KUKA KRL program: EPS_2_251806_MH47A_A_20260213065144.src

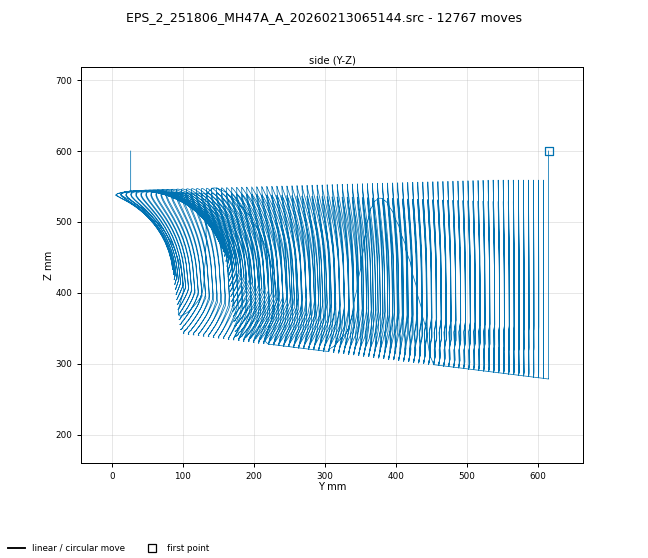
[picture p0: tool path of EPS_2_251806_MH47A_A_20260213065144.src, 12767 of 12769 moves have a stored position in this frame; points joined in program order, loops and branches not executed]
&ACCESS RVP
&REL 4
&COMMENT QRS 19112012
&PARAM EDITMASK = *
DEF PART()
EXT BAS (BAS_COMMAND :IN,REAL :IN )
INT I
BAS (#INITMOV,0 )

;KUKA QRS Post kuka4.cps  Date:22-06-2017 !

File_ID=3034

QRS_PRE_INIT()

;Init var - Until changes are made in qrs_pre_init
Outlet_Square_prg=0
Inlet_1_Square_prg=0
Inlet_2_Square_prg=0
Inlet_3_Square_prg=0
Inlet_4_Square_prg=0
Inlet_5_Square_prg=0

Outlet_1={X 0.000, Y 535.490, Z 458.500, B 0.000, E1 0.000 }
Inlet_1={X 0.000, Y 537.630, Z 428.500, B 0.000, E1 194.000 }
Outlet_1_type=201
Inlet_1_type=201
;QRS#1=Sidecore dimensions
;QRS#2=200-8" PVC SDR 35
;QRS#3=200-8" PVC SDR 35
;QRS#4=
;QRS#5=
;QRS#6=
;QRS#7=
;QRS#8=
;QRS#9=12-08 PSX
;QRS#10=12-08 PSX
;QRS#11=
;QRS#12=
;QRS#13=
;QRS#14=
;QRS#15=
;QRS#16=1220x127x838 2,75'
;QRS#17=EPS Height
;QRS#18=559
;QRS#19=*
;QRS#20= UPDATED VERSION 22-06-2017
;QRS#21=*
Outlet_Square=0100
Inlet_1_Square=0100
Inlet_2_Square=0
Inlet_3_Square=0
Inlet_4_Square=0
Inlet_5_Square=0
Mill_Square=1
Outlet_Square_Prg=204
Inlet_1_Square_prg=204

QRS_INIT()

$ADVANCE=5

; T1
PTP {E1 173.619,E2 173.619}
PTP {X 0,Y 615.497,A -85,B 0,C 180,E1 173.619,E2 173.619,E3 0,E4 0,E5 0,E6 0}
QRS_SPEED_INIT()
LIN {X 0,Y 615.497,Z 600,A -85,B 0,C 180,E1 173.619,E2 173.619,E3 0,E4 0,E5 0,E6 0} C_VEL
LIN {X 0,Y 615.497,Z 288.877,A -85,B 0,C 180,E1 173.619,E2 173.619} C_VEL
LIN {X 0,Y 615.497,Z 280.697,A -85,B 0,C 180,E1 173.619,E2 173.619} C_VEL
LIN {X 0,Y 615.476,Z 278.697,A -85,B 0,C 180,E1 173.433,E2 173.433} C_VEL
LIN {X 0,Y 615.451,Z 278.69,A -85,B 0,C 180,E1 170.801,E2 170.801} C_VEL
LIN {X 0,Y 615.482,Z 278.683,A -85,B 0,C 180,E1 168.139,E2 168.139} C_VEL
LIN {X 0,Y 615.489,Z 278.698,A -85,B 0,C 180,E1 165.451,E2 165.451} C_VEL
LIN {X 0,Y 615.453,Z 278.694,A -85,B 0,C 180,E1 162.729,E2 162.729} C_VEL
LIN {X 0,Y 615.455,Z 278.693,A -85,B 0,C 180,E1 160.661,E2 160.661} C_VEL
LIN {X 0,Y 615.455,Z 278.693,A -85,B 0,C 180,E1 158.567,E2 158.567} C_VEL
LIN {X 0,Y 615.458,Z 278.687,A -85,B 0,C 180,E1 155.998,E2 155.998} C_VEL
LIN {X 0,Y 615.483,Z 278.683,A -85,B 0,C 180,E1 153.556,E2 153.556} C_VEL
LIN {X 0,Y 615.475,Z 278.699,A -85,B 0,C 180,E1 150.593,E2 150.593} C_VEL
LIN {X 0,Y 615.462,Z 278.695,A -85,B 0,C 180,E1 148.313,E2 148.313} C_VEL
LIN {X 0,Y 615.451,Z 278.692,A -85,B 0,C 180,E1 145.976,E2 145.976} C_VEL
LIN {X 0,Y 615.455,Z 278.688,A -85,B 0,C 180,E1 143.573,E2 143.573} C_VEL
LIN {X 0,Y 615.494,Z 278.683,A -85,B 0,C 180,E1 140.938,E2 140.938} C_VEL
LIN {X 0,Y 615.491,Z 278.693,A -85,B 0,C 180,E1 138.527,E2 138.527} C_VEL
LIN {X 0,Y 615.46,Z 278.696,A -85,B 0,C 180,E1 135.848,E2 135.848} C_VEL
LIN {X 0,Y 615.452,Z 278.689,A -85,B 0,C 180,E1 133.248,E2 133.248} C_VEL
LIN {X 0,Y 615.488,Z 278.683,A -85,B 0,C 180,E1 130.607,E2 130.607} C_VEL
LIN {X 0,Y 615.487,Z 278.698,A -85,B 0,C 180,E1 128.012,E2 128.012} C_VEL
LIN {X 0,Y 615.477,Z 278.698,A -85,B 0,C 180,E1 125.617,E2 125.617} C_VEL
LIN {X 0,Y 615.455,Z 278.694,A -85,B 0,C 180,E1 123.239,E2 123.239} C_VEL
LIN {X 0,Y 615.447,Z 278.691,A -85,B 0,C 180,E1 120.922,E2 120.922} C_VEL
LIN {X 0,Y 615.462,Z 278.686,A -85,B 0,C 180,E1 118.446,E2 118.446} C_VEL
LIN {X 0,Y 615.491,Z 278.696,A -85,B 0,C 180,E1 115.57,E2 115.57} C_VEL
LIN {X 0,Y 615.455,Z 278.694,A -85,B 0,C 180,E1 112.846,E2 112.846} C_VEL
LIN {X 0,Y 615.449,Z 278.691,A -85,B 0,C 180,E1 110.548,E2 110.548} C_VEL
LIN {X 0,Y 615.47,Z 278.685,A -85,B 0,C 180,E1 107.958,E2 107.958} C_VEL
LIN {X 0,Y 615.493,Z 278.694,A -85,B 0,C 180,E1 105.226,E2 105.226} C_VEL
LIN {X 0,Y 615.459,Z 278.695,A -85,B 0,C 180,E1 102.531,E2 102.531} C_VEL
LIN {X 0,Y 615.465,Z 278.696,A -85,B 0,C 180,E1 100.528,E2 100.528} C_VEL
LIN {X 0,Y 615.472,Z 278.697,A -85,B 0,C 180,E1 98.537,E2 98.537} C_VEL
LIN {X 0,Y 615.448,Z 278.69,A -85,B 0,C 180,E1 95.899,E2 95.899} C_VEL
LIN {X 0,Y 615.489,Z 278.782,A -85,B 0,C 180,E1 95.201,E2 95.201} C_VEL
LIN {X 0,Y 615.493,Z 296.487,A -85,B 0,C 180,E1 92.291,E2 92.291} C_VEL
LIN {X 0,Y 615.474,Z 313.65,A -85,B 0,C 180,E1 89.51,E2 89.51} C_VEL
LIN {X 0,Y 615.497,Z 317.957,A -85,B 0,C 180,E1 88.815,E2 88.815} C_VEL
LIN {X 0,Y 615.476,Z 424.728,A -85,B 0,C 180,E1 87.546,E2 87.546} C_VEL
LIN {X 0,Y 615.474,Z 437.838,A -85,B 0,C 180,E1 87.26,E2 87.26} C_VEL
LIN {X 0,Y 615.498,Z 450.38,A -85,B 0,C 180,E1 86.851,E2 86.851} C_VEL
LIN {X 0,Y 615.484,Z 462.433,A -85,B 0,C 180,E1 86.318,E2 86.318} C_VEL
LIN {X 0,Y 615.494,Z 473.824,A -85,B 0,C 180,E1 85.662,E2 85.662} C_VEL
LIN {X 0,Y 615.499,Z 483.003,A -85,B 0,C 180,E1 85.006,E2 85.006} C_VEL
LIN {X 0,Y 615.497,Z 491.611,A -85,B 0,C 180,E1 84.267,E2 84.267} C_VEL
LIN {X 0,Y 615.494,Z 499.888,A -85,B 0,C 180,E1 83.416,E2 83.416} C_VEL
LIN {X 0,Y 615.49,Z 507.472,A -85,B 0,C 180,E1 82.455,E2 82.455} C_VEL
LIN {X 0,Y 615.496,Z 513.737,A -85,B 0,C 180,E1 81.464,E2 81.464} C_VEL
LIN {X 0,Y 615.497,Z 518.737,A -85,B 0,C 180,E1 80.471,E2 80.471} C_VEL
LIN {X 0,Y 615.497,Z 522.611,A -85,B 0,C 180,E1 79.474,E2 79.474} C_VEL
LIN {X 0,Y 615.497,Z 524.605,A -85,B 0,C 180,E1 78.808,E2 78.808} C_VEL
LIN {X 0,Y 615.495,Z 526.183,A -85,B 0,C 180,E1 78.14,E2 78.14} C_VEL
LIN {X 0,Y 615.496,Z 527.336,A -85,B 0,C 180,E1 77.471,E2 77.471} C_VEL
LIN {X 0,Y 615.495,Z 528.353,A -85,B 0,C 180,E1 76.127,E2 76.127} C_VEL
LIN {X 0,Y 615.497,Z 528.272,A -85,B 0,C 180,E1 75.452,E2 75.452} C_VEL
LIN {X 0,Y 615.494,Z 527.732,A -85,B 0,C 180,E1 74.775,E2 74.775} C_VEL
LIN {X 0,Y 615.494,Z 525.742,A -85,B 0,C 180,E1 73.567,E2 73.567} C_VEL
LIN {X 0,Y 615.496,Z 522.457,A -85,B 0,C 180,E1 72.388,E2 72.388} C_VEL
LIN {X 0,Y 615.497,Z 518.375,A -85,B 0,C 180,E1 71.355,E2 71.355} C_VEL
LIN {X 0,Y 615.497,Z 511.947,A -85,B 0,C 180,E1 70.142,E2 70.142} C_VEL
LIN {X 0,Y 615.497,Z 504.808,A -85,B 0,C 180,E1 69.095,E2 69.095} C_VEL
LIN {X 0,Y 615.499,Z 497.411,A -85,B 0,C 180,E1 68.218,E2 68.218} C_VEL
LIN {X 0,Y 615.496,Z 487.591,A -85,B 0,C 180,E1 67.28,E2 67.28} C_VEL
LIN {X 0,Y 615.493,Z 478.076,A -85,B 0,C 180,E1 66.534,E2 66.534} C_VEL
LIN {X 0,Y 615.484,Z 467.445,A -85,B 0,C 180,E1 65.86,E2 65.86} C_VEL
LIN {X 0,Y 615.494,Z 455.76,A -85,B 0,C 180,E1 65.28,E2 65.28} C_VEL
LIN {X 0,Y 615.481,Z 442.758,A -85,B 0,C 180,E1 64.794,E2 64.794} C_VEL
LIN {X 0,Y 615.472,Z 430.437,A -85,B 0,C 180,E1 64.47,E2 64.47} C_VEL
LIN {X 0,Y 615.476,Z 417.236,A -85,B 0,C 180,E1 64.262,E2 64.262} C_VEL
LIN {X 0,Y 615.496,Z 317.894,A -85,B 0,C 180,E1 63.085,E2 63.085} C_VEL
LIN {X 0,Y 615.476,Z 300.108,A -85,B 0,C 180,E1 60.207,E2 60.207} C_VEL
LIN {X 0,Y 615.495,Z 283.831,A -85,B 0,C 180,E1 57.544,E2 57.544} C_VEL
LIN {X 0,Y 615.443,Z 278.695,A -85,B 0,C 180,E1 56.69,E2 56.69} C_VEL
LIN {X 0,Y 615.442,Z 278.691,A -85,B 0,C 180,E1 54.172,E2 54.172} C_VEL
LIN {X 0,Y 615.451,Z 278.69,A -85,B 0,C 180,E1 51.93,E2 51.93} C_VEL
LIN {X 0,Y 615.49,Z 278.69,A -85,B 0,C 180,E1 49.395,E2 49.395} C_VEL
LIN {X 0,Y 615.469,Z 278.698,A -85,B 0,C 180,E1 46.755,E2 46.755} C_VEL
LIN {X 0,Y 615.431,Z 278.695,A -85,B 0,C 180,E1 44.155,E2 44.155} C_VEL
LIN {X 0,Y 615.429,Z 278.695,A -85,B 0,C 180,E1 42.075,E2 42.075} C_VEL
LIN {X 0,Y 615.429,Z 278.694,A -85,B 0,C 180,E1 39.755,E2 39.755} C_VEL
LIN {X 0,Y 615.458,Z 278.692,A -85,B 0,C 180,E1 37.244,E2 37.244} C_VEL
LIN {X 0,Y 615.498,Z 278.697,A -85,B 0,C 180,E1 34.704,E2 34.704} C_VEL
LIN {X 0,Y 615.468,Z 278.699,A -85,B 0,C 180,E1 32.33,E2 32.33} C_VEL
LIN {X 0,Y 615.421,Z 278.698,A -85,B 0,C 180,E1 29.786,E2 29.786} C_VEL
LIN {X 0,Y 615.434,Z 278.699,A -85,B 0,C 180,E1 27.918,E2 27.918} C_VEL
LIN {X 0,Y 615.418,Z 278.697,A -85,B 0,C 180,E1 25.557,E2 25.557} C_VEL
LIN {X 0,Y 615.419,Z 278.698,A -85,B 0,C 180,E1 23.559,E2 23.559} C_VEL
LIN {X 0,Y 615.415,Z 278.698,A -85,B 0,C 180,E1 21.434,E2 21.434} C_VEL
LIN {X 0,Y 615.413,Z 278.698,A -85,B 0,C 180,E1 19.34,E2 19.34} C_VEL
LIN {X 0,Y 615.411,Z 278.699,A -85,B 0,C 180,E1 17.273,E2 17.273} C_VEL
LIN {X 0,Y 615.41,Z 278.699,A -85,B 0,C 180,E1 15.228,E2 15.228} C_VEL
LIN {X 0,Y 615.411,Z 278.699,A -85,B 0,C 180,E1 13.203,E2 13.203} C_VEL
LIN {X 0,Y 615.404,Z 278.699,A -85,B 0,C 180,E1 10.853,E2 10.853} C_VEL
LIN {X 0,Y 615.415,Z 278.7,A -85,B 0,C 180,E1 9.2,E2 9.2} C_VEL
LIN {X 0,Y 615.421,Z 278.7,A -85,B 0,C 180,E1 7.216,E2 7.216} C_VEL
LIN {X 0,Y 615.43,Z 278.7,A -85,B 0,C 180,E1 5.242,E2 5.242} C_VEL
LIN {X 0,Y 615.443,Z 278.699,A -85,B 0,C 180,E1 3.273,E2 3.273} C_VEL
LIN {X 0,Y 615.406,Z 278.699,A -85,B 0,C 180,E1 0.654,E2 0.654} C_VEL
LIN {X 0,Y 615.411,Z 278.698,A -85,B 0,C 180,E1 -1.309,E2 -1.309} C_VEL
LIN {X 0,Y 615.418,Z 278.698,A -85,B 0,C 180,E1 -3.273,E2 -3.273} C_VEL
LIN {X 0,Y 615.426,Z 278.697,A -85,B 0,C 180,E1 -5.242,E2 -5.242} C_VEL
LIN {X 0,Y 615.437,Z 278.696,A -85,B 0,C 180,E1 -7.216,E2 -7.216} C_VEL
LIN {X 0,Y 615.448,Z 278.695,A -85,B 0,C 180,E1 -9.2,E2 -9.2} C_VEL
LIN {X 0,Y 615.459,Z 278.695,A -85,B 0,C 180,E1 -11.194,E2 -11.194} C_VEL
LIN {X 0,Y 615.417,Z 278.696,A -85,B 0,C 180,E1 -13.91,E2 -13.91} C_VEL
LIN {X 0,Y 615.418,Z 278.696,A -85,B 0,C 180,E1 -15.907,E2 -15.907} C_VEL
LIN {X 0,Y 615.422,Z 278.695,A -85,B 0,C 180,E1 -17.959,E2 -17.959} C_VEL
LIN {X 0,Y 615.422,Z 278.695,A -85,B 0,C 180,E1 -20.035,E2 -20.035} C_VEL
LIN {X 0,Y 615.424,Z 278.696,A -85,B 0,C 180,E1 -22.334,E2 -22.334} C_VEL
LIN {X 0,Y 615.469,Z 278.699,A -85,B 0,C 180,E1 -24.993,E2 -24.993} C_VEL
LIN {X 0,Y 615.455,Z 278.691,A -85,B 0,C 180,E1 -27.917,E2 -27.917} C_VEL
LIN {X 0,Y 615.442,Z 278.692,A -85,B 0,C 180,E1 -30.163,E2 -30.163} C_VEL
LIN {X 0,Y 615.433,Z 278.693,A -85,B 0,C 180,E1 -32.461,E2 -32.461} C_VEL
LIN {X 0,Y 615.432,Z 278.695,A -85,B 0,C 180,E1 -34.819,E2 -34.819} C_VEL
LIN {X 0,Y 615.458,Z 278.697,A -85,B 0,C 180,E1 -37.244,E2 -37.244} C_VEL
LIN {X 0,Y 615.495,Z 278.686,A -85,B 0,C 180,E1 -40.091,E2 -40.091} C_VEL
LIN {X 0,Y 615.468,Z 278.688,A -85,B 0,C 180,E1 -42.355,E2 -42.355} C_VEL
LIN {X 0,Y 615.441,Z 278.691,A -85,B 0,C 180,E1 -44.928,E2 -44.928} C_VEL
LIN {X 0,Y 615.443,Z 278.691,A -85,B 0,C 180,E1 -46.957,E2 -46.957} C_VEL
LIN {X 0,Y 615.447,Z 278.694,A -85,B 0,C 180,E1 -49.391,E2 -49.391} C_VEL
LIN {X 0,Y 615.48,Z 278.703,A -85,B 0,C 180,E1 -51.989,E2 -51.989} C_VEL
LIN {X 0,Y 615.493,Z 278.69,A -85,B 0,C 180,E1 -54.386,E2 -54.386} C_VEL
LIN {X 0,Y 615.485,Z 278.684,A -85,B 0,C 180,E1 -56.765,E2 -56.765} C_VEL
LIN {X 0,Y 615.468,Z 278.685,A -85,B 0,C 180,E1 -59.08,E2 -59.08} C_VEL
LIN {X 0,Y 615.45,Z 278.69,A -85,B 0,C 180,E1 -61.557,E2 -61.557} C_VEL
LIN {X 0,Y 615.451,Z 278.689,A -85,B 0,C 180,E1 -63.555,E2 -63.555} C_VEL
LIN {X 0,Y 615.459,Z 278.694,A -85,B 0,C 180,E1 -65.998,E2 -65.998} C_VEL
LIN {X 0,Y 615.454,Z 278.772,A -85,B 0,C 180,E1 -67.838,E2 -67.838} C_VEL
LIN {X 0,Y 615.483,Z 297.825,A -85,B 0,C 180,E1 -70.489,E2 -70.489} C_VEL
LIN {X 0,Y 615.496,Z 319.19,A -85,B 0,C 180,E1 -73.414,E2 -73.414} C_VEL
LIN {X 0,Y 615.486,Z 340.532,A -85,B 0,C 180,E1 -76.295,E2 -76.295} C_VEL
LIN {X 0,Y 615.476,Z 346.648,A -85,B 0,C 180,E1 -77.114,E2 -77.114} C_VEL
LIN {X 0,Y 615.488,Z 454.868,A -85,B 0,C 180,E1 -78.411,E2 -78.411} C_VEL
LIN {X 0,Y 615.493,Z 467.368,A -85,B 0,C 180,E1 -78.683,E2 -78.683} C_VEL
LIN {X 0,Y 615.492,Z 480.562,A -85,B 0,C 180,E1 -79.111,E2 -79.111} C_VEL
LIN {X 0,Y 615.489,Z 492.49,A -85,B 0,C 180,E1 -79.64,E2 -79.64} C_VEL
LIN {X 0,Y 615.478,Z 504.007,A -85,B 0,C 180,E1 -80.304,E2 -80.304} C_VEL
LIN {X 0,Y 615.498,Z 513.229,A -85,B 0,C 180,E1 -80.968,E2 -80.968} C_VEL
LIN {X 0,Y 615.498,Z 521.009,A -85,B 0,C 180,E1 -81.63,E2 -81.63} C_VEL
LIN {X 0,Y 615.497,Z 530.612,A -85,B 0,C 180,E1 -82.62,E2 -82.62} C_VEL
LIN {X 0,Y 615.49,Z 538.208,A -85,B 0,C 180,E1 -83.609,E2 -83.609} C_VEL
LIN {X 0,Y 615.498,Z 545.208,A -85,B 0,C 180,E1 -84.76,E2 -84.76} C_VEL
LIN {X 0,Y 615.493,Z 549.854,A -85,B 0,C 180,E1 -85.744,E2 -85.744} C_VEL
LIN {X 0,Y 615.496,Z 553.4,A -85,B 0,C 180,E1 -86.728,E2 -86.728} C_VEL
LIN {X 0,Y 615.497,Z 555.234,A -85,B 0,C 180,E1 -87.383,E2 -87.383} C_VEL
LIN {X 0,Y 615.496,Z 556.609,A -85,B 0,C 180,E1 -88.038,E2 -88.038} C_VEL
LIN {X 0,Y 615.496,Z 558.174,A -85,B 0,C 180,E1 -89.346,E2 -89.346} C_VEL
LIN {X 0,Y 615.494,Z 558.389,A -85,B 0,C 180,E1 -90.001,E2 -90.001} C_VEL
LIN {X 0,Y 615.496,Z 557.579,A -85,B 0,C 180,E1 -91.309,E2 -91.309} C_VEL
LIN {X 0,Y 615.496,Z 556.607,A -85,B 0,C 180,E1 -91.964,E2 -91.964} C_VEL
LIN {X 0,Y 615.497,Z 555.231,A -85,B 0,C 180,E1 -92.618,E2 -92.618} C_VEL
LIN {X 0,Y 615.496,Z 552.348,A -85,B 0,C 180,E1 -93.601,E2 -93.601} C_VEL
LIN {X 0,Y 615.498,Z 548.439,A -85,B 0,C 180,E1 -94.585,E2 -94.585} C_VEL
LIN {X 0,Y 615.499,Z 543.402,A -85,B 0,C 180,E1 -95.57,E2 -95.57} C_VEL
LIN {X 0,Y 615.489,Z 536.916,A -85,B 0,C 180,E1 -96.577,E2 -96.577} C_VEL
LIN {X 0,Y 615.497,Z 529.128,A -85,B 0,C 180,E1 -97.546,E2 -97.546} C_VEL
LIN {X 0,Y 615.498,Z 519.251,A -85,B 0,C 180,E1 -98.537,E2 -98.537} C_VEL
LIN {X 0,Y 615.492,Z 507.703,A -85,B 0,C 180,E1 -99.448,E2 -99.448} C_VEL
LIN {X 0,Y 615.48,Z 497.146,A -85,B 0,C 180,E1 -100.112,E2 -100.112} C_VEL
LIN {X 0,Y 615.496,Z 484.985,A -85,B 0,C 180,E1 -100.708,E2 -100.708} C_VEL
LIN {X 0,Y 615.489,Z 472.929,A -85,B 0,C 180,E1 -101.155,E2 -101.155} C_VEL
LIN {X 0,Y 615.491,Z 460.391,A -85,B 0,C 180,E1 -101.485,E2 -101.485} C_VEL
LIN {X 0,Y 615.487,Z 447.114,A -85,B 0,C 180,E1 -101.694,E2 -101.694} C_VEL
LIN {X 0,Y 615.475,Z 346.639,A -85,B 0,C 180,E1 -102.887,E2 -102.887} C_VEL
LIN {X 0,Y 615.496,Z 325.461,A -85,B 0,C 180,E1 -105.735,E2 -105.735} C_VEL
LIN {X 0,Y 615.486,Z 304.104,A -85,B 0,C 180,E1 -108.647,E2 -108.647} C_VEL
LIN {X 0,Y 615.497,Z 283.977,A -85,B 0,C 180,E1 -111.432,E2 -111.432} C_VEL
LIN {X 0,Y 615.454,Z 278.69,A -85,B 0,C 180,E1 -112.188,E2 -112.188} C_VEL
LIN {X 0,Y 615.492,Z 278.682,A -85,B 0,C 180,E1 -114.992,E2 -114.992} C_VEL
LIN {X 0,Y 615.478,Z 278.697,A -85,B 0,C 180,E1 -117.916,E2 -117.916} C_VEL
LIN {X 0,Y 615.465,Z 278.695,A -85,B 0,C 180,E1 -120.162,E2 -120.162} C_VEL
LIN {X 0,Y 615.455,Z 278.692,A -85,B 0,C 180,E1 -122.46,E2 -122.46} C_VEL
LIN {X 0,Y 615.456,Z 278.688,A -85,B 0,C 180,E1 -124.818,E2 -124.818} C_VEL
LIN {X 0,Y 615.476,Z 278.683,A -85,B 0,C 180,E1 -127.243,E2 -127.243} C_VEL
LIN {X 0,Y 615.494,Z 278.697,A -85,B 0,C 180,E1 -130.089,E2 -130.089} C_VEL
LIN {X 0,Y 615.491,Z 278.699,A -85,B 0,C 180,E1 -132.353,E2 -132.353} C_VEL
LIN {X 0,Y 615.45,Z 278.691,A -85,B 0,C 180,E1 -135.072,E2 -135.072} C_VEL
LIN {X 0,Y 615.496,Z 278.682,A -85,B 0,C 180,E1 -137.919,E2 -137.919} C_VEL
LIN {X 0,Y 615.49,Z 278.69,A -85,B 0,C 180,E1 -140.25,E2 -140.25} C_VEL
LIN {X 0,Y 615.463,Z 278.695,A -85,B 0,C 180,E1 -143.067,E2 -143.067} C_VEL
LIN {X 0,Y 615.455,Z 278.693,A -85,B 0,C 180,E1 -145.304,E2 -145.304} C_VEL
LIN {X 0,Y 615.454,Z 278.689,A -85,B 0,C 180,E1 -147.675,E2 -147.675} C_VEL
LIN {X 0,Y 615.482,Z 278.683,A -85,B 0,C 180,E1 -150.207,E2 -150.207} C_VEL
LIN {X 0,Y 615.494,Z 278.697,A -85,B 0,C 180,E1 -152.954,E2 -152.954} C_VEL
LIN {X 0,Y 615.452,Z 278.693,A -85,B 0,C 180,E1 -155.726,E2 -155.726} C_VEL
LIN {X 0,Y 615.453,Z 278.692,A -85,B 0,C 180,E1 -157.862,E2 -157.862} C_VEL
LIN {X 0,Y 615.451,Z 278.692,A -85,B 0,C 180,E1 -159.966,E2 -159.966} C_VEL
LIN {X 0,Y 615.453,Z 278.691,A -85,B 0,C 180,E1 -162.042,E2 -162.042} C_VEL
LIN {X 0,Y 615.483,Z 278.682,A -85,B 0,C 180,E1 -164.774,E2 -164.774} C_VEL
LIN {X 0,Y 615.489,Z 278.696,A -85,B 0,C 180,E1 -167.47,E2 -167.47} C_VEL
LIN {X 0,Y 615.46,Z 278.694,A -85,B 0,C 180,E1 -170.137,E2 -170.137} C_VEL
LIN {X 0,Y 615.458,Z 278.687,A -85,B 0,C 180,E1 -172.784,E2 -172.784} C_VEL
LIN {X 0,Y 615.495,Z 278.684,A -85,B 0,C 180,E1 -175.415,E2 -175.415} C_VEL
LIN {X 0,Y 615.499,Z 278.7,A -85,B 0,C 180,E1 -178.037,E2 -178.037} C_VEL
LIN {X 0,Y 615.454,Z 278.693,A -85,B 0,C 180,E1 -180.654,E2 -180.654} C_VEL
LIN {X 0,Y 615.463,Z 278.686,A -85,B 0,C 180,E1 -183.273,E2 -183.273} C_VEL
LIN {X 0,Y 615.493,Z 278.686,A -85,B 0,C 180,E1 -185.898,E2 -185.898} C_VEL
LIN {X 0,Y 615.476,Z 278.697,A -85,B 0,C 180,E1 -186.567,E2 -186.567} C_VEL
LIN {X 0,Y 614.782,Z 278.836,A -85,B 0,C 180,E1 -187.113,E2 -187.113} C_VEL
LIN {X 0,Y 611.932,Z 279.257,A -85,B 0,C 180,E1 -187.999,E2 -187.999} C_VEL
LIN {X 0,Y 609.544,Z 279.564,A -85,B 0,C 180,E1 -188.711,E2 -188.711} C_VEL
LIN {X 0,Y 608.523,Z 279.679,A -85,B 0,C 180,E1 -189.261,E2 -189.261} C_VEL
LIN {X 0,Y 608.442,Z 279.687,A -85,B 0,C 180,E1 -189.447,E2 -189.447} C_VEL
LIN {X 0,Y 608.461,Z 279.687,A -85,B 0,C 180,E1 -192,E2 -192} C_VEL
LIN {X 0,Y 608.47,Z 279.695,A -85,B 0,C 180,E1 -194.72,E2 -194.72} C_VEL
LIN {X 0,Y 608.427,Z 279.69,A -85,B 0,C 180,E1 -197.477,E2 -197.477} C_VEL
LIN {X 0,Y 608.43,Z 279.69,A -85,B 0,C 180,E1 -199.571,E2 -199.571} C_VEL
LIN {X 0,Y 608.445,Z 279.688,A -85,B 0,C 180,E1 -201.692,E2 -201.692} C_VEL
LIN {X 0,Y 608.454,Z 279.689,A -85,B 0,C 180,E1 -204.571,E2 -204.571} C_VEL
LIN {X 0,Y 608.436,Z 279.693,A -85,B 0,C 180,E1 -207.518,E2 -207.518} C_VEL
LIN {X 0,Y 608.421,Z 279.691,A -85,B 0,C 180,E1 -209.963,E2 -209.963} C_VEL
LIN {X 0,Y 608.446,Z 279.687,A -85,B 0,C 180,E1 -212.52,E2 -212.52} C_VEL
LIN {X 0,Y 608.444,Z 279.695,A -85,B 0,C 180,E1 -215.277,E2 -215.277} C_VEL
LIN {X 0,Y 608.453,Z 279.694,A -85,B 0,C 180,E1 -217.747,E2 -217.747} C_VEL
LIN {X 0,Y 608.434,Z 279.69,A -85,B 0,C 180,E1 -220.327,E2 -220.327} C_VEL
LIN {X 0,Y 608.483,Z 279.686,A -85,B 0,C 180,E1 -223.31,E2 -223.31} C_VEL
LIN {X 0,Y 608.465,Z 279.691,A -85,B 0,C 180,E1 -226.13,E2 -226.13} C_VEL
LIN {X 0,Y 608.423,Z 279.69,A -85,B 0,C 180,E1 -228.82,E2 -228.82} C_VEL
LIN {X 0,Y 608.465,Z 279.69,A -85,B 0,C 180,E1 -231.76,E2 -231.76} C_VEL
LIN {X 0,Y 608.428,Z 279.692,A -85,B 0,C 180,E1 -234.721,E2 -234.721} C_VEL
LIN {X 0,Y 608.439,Z 279.688,A -85,B 0,C 180,E1 -237.119,E2 -237.119} C_VEL
LIN {X 0,Y 608.475,Z 279.688,A -85,B 0,C 180,E1 -240.027,E2 -240.027} C_VEL
LIN {X 0,Y 608.462,Z 279.691,A -85,B 0,C 180,E1 -242.796,E2 -242.796} C_VEL
LIN {X 0,Y 608.433,Z 279.689,A -85,B 0,C 180,E1 -245.428,E2 -245.428} C_VEL
LIN {X 0,Y 608.464,Z 279.689,A -85,B 0,C 180,E1 -248.308,E2 -248.308} C_VEL
LIN {X 0,Y 608.45,Z 279.69,A -85,B 0,C 180,E1 -251.29,E2 -251.29} C_VEL
LIN {X 0,Y 608.437,Z 279.688,A -85,B 0,C 180,E1 -253.905,E2 -253.905} C_VEL
LIN {X 0,Y 608.461,Z 279.689,A -85,B 0,C 180,E1 -256.643,E2 -256.643} C_VEL
LIN {X 0,Y 608.452,Z 279.694,A -85,B 0,C 180,E1 -259.349,E2 -259.349} C_VEL
LIN {X 0,Y 608.447,Z 279.696,A -85,B 0,C 180,E1 -261.363,E2 -261.363} C_VEL
LIN {X 0,Y 608.427,Z 279.691,A -85,B 0,C 180,E1 -264.032,E2 -264.032} C_VEL
LIN {X 0,Y 608.484,Z 279.852,A -85,B 0,C 180,E1 -264.739,E2 -264.739} C_VEL
LIN {X 0,Y 608.508,Z 297.604,A -85,B 0,C 180,E1 -267.683,E2 -267.683} C_VEL
LIN {X 0,Y 608.448,Z 314.835,A -85,B 0,C 180,E1 -270.496,E2 -270.496} C_VEL
LIN {X 0,Y 608.473,Z 318.148,A -85,B 0,C 180,E1 -271.033,E2 -271.033} C_VEL
LIN {X 0,Y 608.539,Z 425.77,A -85,B 0,C 180,E1 -272.337,E2 -272.337} C_VEL
LIN {X 0,Y 608.527,Z 439.312,A -85,B 0,C 180,E1 -272.647,E2 -272.647} C_VEL
LIN {X 0,Y 608.538,Z 451.522,A -85,B 0,C 180,E1 -273.061,E2 -273.061} C_VEL
LIN {X 0,Y 608.5,Z 462.529,A -85,B 0,C 180,E1 -273.559,E2 -273.559} C_VEL
LIN {X 0,Y 608.504,Z 473.975,A -85,B 0,C 180,E1 -274.222,E2 -274.222} C_VEL
LIN {X 0,Y 608.473,Z 483.226,A -85,B 0,C 180,E1 -274.886,E2 -274.886} C_VEL
LIN {X 0,Y 608.47,Z 491.883,A -85,B 0,C 180,E1 -275.634,E2 -275.634} C_VEL
LIN {X 0,Y 608.466,Z 500.297,A -85,B 0,C 180,E1 -276.504,E2 -276.504} C_VEL
LIN {X 0,Y 608.443,Z 507.856,A -85,B 0,C 180,E1 -277.466,E2 -277.466} C_VEL
LIN {X 0,Y 608.456,Z 513.22,A -85,B 0,C 180,E1 -278.301,E2 -278.301} C_VEL
LIN {X 0,Y 608.432,Z 518.486,A -85,B 0,C 180,E1 -279.306,E2 -279.306} C_VEL
LIN {X 0,Y 608.438,Z 522.578,A -85,B 0,C 180,E1 -280.313,E2 -280.313} C_VEL
LIN {X 0,Y 608.425,Z 525.617,A -85,B 0,C 180,E1 -281.324,E2 -281.324} C_VEL
LIN {X 0,Y 608.44,Z 527.102,A -85,B 0,C 180,E1 -282,E2 -282} C_VEL
LIN {X 0,Y 608.44,Z 528.765,A -85,B 0,C 180,E1 -283.356,E2 -283.356} C_VEL
LIN {X 0,Y 608.423,Z 529,A -85,B 0,C 180,E1 -284.038,E2 -284.038} C_VEL
LIN {X 0,Y 608.418,Z 528.773,A -85,B 0,C 180,E1 -284.721,E2 -284.721} C_VEL
LIN {X 0,Y 608.417,Z 528.139,A -85,B 0,C 180,E1 -285.407,E2 -285.407} C_VEL
LIN {X 0,Y 608.424,Z 526.209,A -85,B 0,C 180,E1 -286.515,E2 -286.515} C_VEL
LIN {X 0,Y 608.427,Z 522.404,A -85,B 0,C 180,E1 -287.824,E2 -287.824} C_VEL
LIN {X 0,Y 608.457,Z 518.074,A -85,B 0,C 180,E1 -288.869,E2 -288.869} C_VEL
LIN {X 0,Y 608.437,Z 512.414,A -85,B 0,C 180,E1 -289.922,E2 -289.922} C_VEL
LIN {X 0,Y 608.471,Z 505.226,A -85,B 0,C 180,E1 -290.98,E2 -290.98} C_VEL
LIN {X 0,Y 608.455,Z 497.773,A -85,B 0,C 180,E1 -291.869,E2 -291.869} C_VEL
LIN {X 0,Y 608.471,Z 487.805,A -85,B 0,C 180,E1 -292.826,E2 -292.826} C_VEL
LIN {X 0,Y 608.473,Z 478.339,A -85,B 0,C 180,E1 -293.573,E2 -293.573} C_VEL
LIN {X 0,Y 608.483,Z 467.965,A -85,B 0,C 180,E1 -294.237,E2 -294.237} C_VEL
LIN {X 0,Y 608.512,Z 455.983,A -85,B 0,C 180,E1 -294.841,E2 -294.841} C_VEL
LIN {X 0,Y 608.537,Z 442.955,A -85,B 0,C 180,E1 -295.333,E2 -295.333} C_VEL
LIN {X 0,Y 608.537,Z 430.54,A -85,B 0,C 180,E1 -295.663,E2 -295.663} C_VEL
LIN {X 0,Y 608.533,Z 416.581,A -85,B 0,C 180,E1 -295.883,E2 -295.883} C_VEL
LIN {X 0,Y 608.493,Z 318.135,A -85,B 0,C 180,E1 -297.058,E2 -297.058} C_VEL
LIN {X 0,Y 608.485,Z 300.242,A -85,B 0,C 180,E1 -299.975,E2 -299.975} C_VEL
LIN {X 0,Y 608.506,Z 284.07,A -85,B 0,C 180,E1 -302.646,E2 -302.646} C_VEL
LIN {X 0,Y 608.421,Z 279.693,A -85,B 0,C 180,E1 -303.399,E2 -303.399} C_VEL
LIN {X 0,Y 608.431,Z 279.69,A -85,B 0,C 180,E1 -306.044,E2 -306.044} C_VEL
LIN {X 0,Y 608.432,Z 279.695,A -85,B 0,C 180,E1 -308.59,E2 -308.59} C_VEL
LIN {X 0,Y 608.437,Z 279.693,A -85,B 0,C 180,E1 -311.34,E2 -311.34} C_VEL
LIN {X 0,Y 608.426,Z 279.69,A -85,B 0,C 180,E1 -313.872,E2 -313.872} C_VEL
LIN {X 0,Y 608.474,Z 279.687,A -85,B 0,C 180,E1 -316.689,E2 -316.689} C_VEL
LIN {X 0,Y 608.411,Z 279.695,A -85,B 0,C 180,E1 -319.693,E2 -319.693} C_VEL
LIN {X 0,Y 608.425,Z 279.69,A -85,B 0,C 180,E1 -322.251,E2 -322.251} C_VEL
LIN {X 0,Y 608.454,Z 279.692,A -85,B 0,C 180,E1 -325.092,E2 -325.092} C_VEL
LIN {X 0,Y 608.434,Z 279.692,A -85,B 0,C 180,E1 -327.904,E2 -327.904} C_VEL
LIN {X 0,Y 608.409,Z 279.693,A -85,B 0,C 180,E1 -330.217,E2 -330.217} C_VEL
LIN {X 0,Y 608.402,Z 279.693,A -85,B 0,C 180,E1 -332.48,E2 -332.48} C_VEL
LIN {X 0,Y 608.388,Z 279.694,A -85,B 0,C 180,E1 -334.696,E2 -334.696} C_VEL
LIN {X 0,Y 608.399,Z 279.693,A -85,B 0,C 180,E1 -336.874,E2 -336.874} C_VEL
LIN {X 0,Y 608.446,Z 279.697,A -85,B 0,C 180,E1 -339.725,E2 -339.725} C_VEL
LIN {X 0,Y 608.401,Z 279.694,A -85,B 0,C 180,E1 -342.522,E2 -342.522} C_VEL
LIN {X 0,Y 608.418,Z 279.692,A -85,B 0,C 180,E1 -344.593,E2 -344.593} C_VEL
LIN {X 0,Y 608.408,Z 279.694,A -85,B 0,C 180,E1 -346.642,E2 -346.642} C_VEL
LIN {X 0,Y 608.375,Z 279.696,A -85,B 0,C 180,E1 -349.085,E2 -349.085} C_VEL
LIN {X 0,Y 608.388,Z 279.695,A -85,B 0,C 180,E1 -351.363,E2 -351.363} C_VEL
LIN {X 0,Y 608.438,Z 279.695,A -85,B 0,C 180,E1 -354.033,E2 -354.033} C_VEL
LIN {X 0,Y 608.413,Z 279.696,A -85,B 0,C 180,E1 -356.689,E2 -356.689} C_VEL
LIN {X 0,Y 608.387,Z 279.695,A -85,B 0,C 180,E1 -359.338,E2 -359.338} C_VEL
LIN {X 0,Y 608.402,Z 279.693,A -85,B 0,C 180,E1 -361.324,E2 -361.324} C_VEL
LIN {X 0,Y 608.387,Z 279.695,A -85,B 0,C 180,E1 -363.311,E2 -363.311} C_VEL
LIN {X 0,Y 608.407,Z 279.693,A -85,B 0,C 180,E1 -365.303,E2 -365.303} C_VEL
LIN {X 0,Y 608.408,Z 279.693,A -85,B 0,C 180,E1 -367.3,E2 -367.3} C_VEL
LIN {X 0,Y 608.429,Z 279.691,A -85,B 0,C 180,E1 -369.307,E2 -369.307} C_VEL
LIN {X 0,Y 608.419,Z 279.693,A -85,B 0,C 180,E1 -371.325,E2 -371.325} C_VEL
LIN {X 0,Y 608.416,Z 279.691,A -85,B 0,C 180,E1 -374.001,E2 -374.001} C_VEL
LIN {X 0,Y 608.431,Z 279.693,A -85,B 0,C 180,E1 -376.521,E2 -376.521} C_VEL
LIN {X 0,Y 608.428,Z 279.692,A -85,B 0,C 180,E1 -379.572,E2 -379.572} C_VEL
LIN {X 0,Y 608.424,Z 279.691,A -85,B 0,C 180,E1 -382.407,E2 -382.407} C_VEL
LIN {X 0,Y 608.443,Z 279.697,A -85,B 0,C 180,E1 -385.302,E2 -385.302} C_VEL
LIN {X 0,Y 608.433,Z 279.696,A -85,B 0,C 180,E1 -387.519,E2 -387.519} C_VEL
LIN {X 0,Y 608.431,Z 279.691,A -85,B 0,C 180,E1 -389.967,E2 -389.967} C_VEL
LIN {X 0,Y 608.416,Z 279.691,A -85,B 0,C 180,E1 -392.517,E2 -392.517} C_VEL
LIN {X 0,Y 608.405,Z 279.694,A -85,B 0,C 180,E1 -394.901,E2 -394.901} C_VEL
LIN {X 0,Y 608.458,Z 279.694,A -85,B 0,C 180,E1 -397.747,E2 -397.747} C_VEL
LIN {X 0,Y 608.437,Z 279.69,A -85,B 0,C 180,E1 -400.329,E2 -400.329} C_VEL
LIN {X 0,Y 608.442,Z 279.689,A -85,B 0,C 180,E1 -402.334,E2 -402.334} C_VEL
LIN {X 0,Y 608.42,Z 279.69,A -85,B 0,C 180,E1 -404.8,E2 -404.8} C_VEL
LIN {X 0,Y 608.413,Z 279.692,A -85,B 0,C 180,E1 -407.038,E2 -407.038} C_VEL
LIN {X 0,Y 608.449,Z 279.694,A -85,B 0,C 180,E1 -409.698,E2 -409.698} C_VEL
LIN {X 0,Y 608.462,Z 279.692,A -85,B 0,C 180,E1 -412.254,E2 -412.254} C_VEL
LIN {X 0,Y 608.421,Z 279.69,A -85,B 0,C 180,E1 -415.099,E2 -415.099} C_VEL
LIN {X 0,Y 608.43,Z 279.69,A -85,B 0,C 180,E1 -417.483,E2 -417.483} C_VEL
LIN {X 0,Y 608.474,Z 279.695,A -85,B 0,C 180,E1 -420.222,E2 -420.222} C_VEL
LIN {X 0,Y 608.44,Z 279.688,A -85,B 0,C 180,E1 -423.226,E2 -423.226} C_VEL
LIN {X 0,Y 608.43,Z 279.692,A -85,B 0,C 180,E1 -425.858,E2 -425.858} C_VEL
LIN {X 0,Y 608.447,Z 279.739,A -85,B 0,C 180,E1 -427.706,E2 -427.706} C_VEL
LIN {X 0,Y 608.542,Z 295.323,A -85,B 0,C 180,E1 -429.906,E2 -429.906} C_VEL
LIN {X 0,Y 608.524,Z 315.472,A -85,B 0,C 180,E1 -432.7,E2 -432.7} C_VEL
LIN {X 0,Y 608.5,Z 335.621,A -85,B 0,C 180,E1 -435.452,E2 -435.452} C_VEL
LIN {X 0,Y 608.512,Z 347.202,A -85,B 0,C 180,E1 -436.985,E2 -436.985} C_VEL
LIN {X 0,Y 608.541,Z 454.984,A -85,B 0,C 180,E1 -438.277,E2 -438.277} C_VEL
LIN {X 0,Y 608.543,Z 468.241,A -85,B 0,C 180,E1 -438.573,E2 -438.573} C_VEL
LIN {X 0,Y 608.517,Z 480.603,A -85,B 0,C 180,E1 -438.981,E2 -438.981} C_VEL
LIN {X 0,Y 608.513,Z 492.648,A -85,B 0,C 180,E1 -439.52,E2 -439.52} C_VEL
LIN {X 0,Y 608.467,Z 504.207,A -85,B 0,C 180,E1 -440.191,E2 -440.191} C_VEL
LIN {X 0,Y 608.472,Z 513.487,A -85,B 0,C 180,E1 -440.863,E2 -440.863} C_VEL
LIN {X 0,Y 608.487,Z 521.31,A -85,B 0,C 180,E1 -441.532,E2 -441.532} C_VEL
LIN {X 0,Y 608.47,Z 530.966,A -85,B 0,C 180,E1 -442.535,E2 -442.535} C_VEL
LIN {X 0,Y 608.435,Z 538.304,A -85,B 0,C 180,E1 -443.487,E2 -443.487} C_VEL
LIN {X 0,Y 608.45,Z 543.869,A -85,B 0,C 180,E1 -444.366,E2 -444.366} C_VEL
LIN {X 0,Y 608.432,Z 548.953,A -85,B 0,C 180,E1 -445.363,E2 -445.363} C_VEL
LIN {X 0,Y 608.449,Z 552.898,A -85,B 0,C 180,E1 -446.358,E2 -446.358} C_VEL
LIN {X 0,Y 608.425,Z 555.811,A -85,B 0,C 180,E1 -447.352,E2 -447.352} C_VEL
LIN {X 0,Y 608.441,Z 557.202,A -85,B 0,C 180,E1 -448.015,E2 -448.015} C_VEL
LIN {X 0,Y 608.438,Z 558.784,A -85,B 0,C 180,E1 -449.339,E2 -449.339} C_VEL
LIN {X 0,Y 608.434,Z 559,A -85,B 0,C 180,E1 -450.001,E2 -450.001} C_VEL
LIN {X 0,Y 608.448,Z 558.183,A -85,B 0,C 180,E1 -451.324,E2 -451.324} C_VEL
LIN {X 0,Y 608.441,Z 557.2,A -85,B 0,C 180,E1 -451.986,E2 -451.986} C_VEL
LIN {X 0,Y 608.425,Z 555.808,A -85,B 0,C 180,E1 -452.649,E2 -452.649} C_VEL
LIN {X 0,Y 608.449,Z 552.894,A -85,B 0,C 180,E1 -453.643,E2 -453.643} C_VEL
LIN {X 0,Y 608.432,Z 548.948,A -85,B 0,C 180,E1 -454.638,E2 -454.638} C_VEL
LIN {X 0,Y 608.437,Z 542.873,A -85,B 0,C 180,E1 -455.801,E2 -455.801} C_VEL
LIN {X 0,Y 608.461,Z 536.231,A -85,B 0,C 180,E1 -456.8,E2 -456.8} C_VEL
LIN {X 0,Y 608.456,Z 527.984,A -85,B 0,C 180,E1 -457.801,E2 -457.801} C_VEL
LIN {X 0,Y 608.469,Z 518.54,A -85,B 0,C 180,E1 -458.72,E2 -458.72} C_VEL
LIN {X 0,Y 608.479,Z 507.922,A -85,B 0,C 180,E1 -459.558,E2 -459.558} C_VEL
LIN {X 0,Y 608.479,Z 497.318,A -85,B 0,C 180,E1 -460.23,E2 -460.23} C_VEL
LIN {X 0,Y 608.512,Z 485.127,A -85,B 0,C 180,E1 -460.832,E2 -460.832} C_VEL
LIN {X 0,Y 608.534,Z 472.866,A -85,B 0,C 180,E1 -461.291,E2 -461.291} C_VEL
LIN {X 0,Y 608.554,Z 460.501,A -85,B 0,C 180,E1 -461.618,E2 -461.618} C_VEL
LIN {X 0,Y 608.558,Z 447.265,A -85,B 0,C 180,E1 -461.829,E2 -461.829} C_VEL
LIN {X 0,Y 608.475,Z 347.099,A -85,B 0,C 180,E1 -463.017,E2 -463.017} C_VEL
LIN {X 0,Y 608.503,Z 326.797,A -85,B 0,C 180,E1 -465.749,E2 -465.749} C_VEL
LIN {X 0,Y 608.506,Z 306.804,A -85,B 0,C 180,E1 -468.497,E2 -468.497} C_VEL
LIN {X 0,Y 608.567,Z 287.758,A -85,B 0,C 180,E1 -471.155,E2 -471.155} C_VEL
LIN {X 0,Y 608.431,Z 279.691,A -85,B 0,C 180,E1 -472.318,E2 -472.318} C_VEL
LIN {X 0,Y 608.441,Z 279.688,A -85,B 0,C 180,E1 -474.572,E2 -474.572} C_VEL
LIN {X 0,Y 608.487,Z 279.685,A -85,B 0,C 180,E1 -477.208,E2 -477.208} C_VEL
LIN {X 0,Y 608.451,Z 279.695,A -85,B 0,C 180,E1 -479.968,E2 -479.968} C_VEL
LIN {X 0,Y 608.447,Z 279.687,A -85,B 0,C 180,E1 -482.881,E2 -482.881} C_VEL
LIN {X 0,Y 608.435,Z 279.689,A -85,B 0,C 180,E1 -485.279,E2 -485.279} C_VEL
LIN {X 0,Y 608.469,Z 279.694,A -85,B 0,C 180,E1 -488.24,E2 -488.24} C_VEL
LIN {X 0,Y 608.431,Z 279.689,A -85,B 0,C 180,E1 -491.179,E2 -491.179} C_VEL
LIN {X 0,Y 608.47,Z 279.687,A -85,B 0,C 180,E1 -493.87,E2 -493.87} C_VEL
LIN {X 0,Y 608.459,Z 279.692,A -85,B 0,C 180,E1 -496.693,E2 -496.693} C_VEL
LIN {X 0,Y 608.438,Z 279.694,A -85,B 0,C 180,E1 -498.822,E2 -498.822} C_VEL
LIN {X 0,Y 608.459,Z 279.685,A -85,B 0,C 180,E1 -501.761,E2 -501.761} C_VEL
LIN {X 0,Y 608.449,Z 279.687,A -85,B 0,C 180,E1 -503.955,E2 -503.955} C_VEL
LIN {X 0,Y 608.453,Z 279.689,A -85,B 0,C 180,E1 -506.328,E2 -506.328} C_VEL
LIN {X 0,Y 608.45,Z 279.695,A -85,B 0,C 180,E1 -508.732,E2 -508.732} C_VEL
LIN {X 0,Y 608.452,Z 279.691,A -85,B 0,C 180,E1 -511.384,E2 -511.384} C_VEL
LIN {X 0,Y 608.428,Z 279.689,A -85,B 0,C 180,E1 -513.963,E2 -513.963} C_VEL
LIN {X 0,Y 608.453,Z 279.691,A -85,B 0,C 180,E1 -516.876,E2 -516.876} C_VEL
LIN {X 0,Y 608.443,Z 279.692,A -85,B 0,C 180,E1 -519.725,E2 -519.725} C_VEL
LIN {X 0,Y 608.428,Z 279.693,A -85,B 0,C 180,E1 -521.827,E2 -521.827} C_VEL
LIN {X 0,Y 608.44,Z 279.692,A -85,B 0,C 180,E1 -523.905,E2 -523.905} C_VEL
LIN {X 0,Y 608.433,Z 279.693,A -85,B 0,C 180,E1 -525.997,E2 -525.997} C_VEL
LIN {X 0,Y 608.442,Z 279.693,A -85,B 0,C 180,E1 -528,E2 -528} C_VEL
LIN {X 0,Y 608.449,Z 279.686,A -85,B 0,C 180,E1 -530.694,E2 -530.694} C_VEL
LIN {X 0,Y 608.482,Z 279.686,A -85,B 0,C 180,E1 -533.367,E2 -533.367} C_VEL
LIN {X 0,Y 608.451,Z 279.697,A -85,B 0,C 180,E1 -536.026,E2 -536.026} C_VEL
LIN {X 0,Y 608.44,Z 279.689,A -85,B 0,C 180,E1 -538.676,E2 -538.676} C_VEL
LIN {X 0,Y 608.458,Z 279.686,A -85,B 0,C 180,E1 -541.324,E2 -541.324} C_VEL
LIN {X 0,Y 608.458,Z 279.692,A -85,B 0,C 180,E1 -543.974,E2 -543.974} C_VEL
LIN {X 0,Y 608.441,Z 279.694,A -85,B 0,C 180,E1 -546.633,E2 -546.633} C_VEL
LIN {X 0,Y 608.448,Z 279.695,A -85,B 0,C 180,E1 -548.636,E2 -548.636} C_VEL
LIN {X 0,Y 608.442,Z 279.687,A -85,B 0,C 180,E1 -549.447,E2 -549.447} C_VEL
LIN {X 0,Y 607.781,Z 279.774,A -85,B 0,C 180,E1 -550,E2 -550} C_VEL
LIN {X 0,Y 604.937,Z 280.129,A -85,B 0,C 180,E1 -550.897,E2 -550.897} C_VEL
LIN {X 0,Y 602.53,Z 280.428,A -85,B 0,C 180,E1 -551.618,E2 -551.618} C_VEL
LIN {X 0,Y 601.493,Z 280.557,A -85,B 0,C 180,E1 -552.175,E2 -552.175} C_VEL
LIN {X 0,Y 601.407,Z 280.568,A -85,B 0,C 180,E1 -552.363,E2 -552.363} C_VEL
LIN {X 0,Y 601.421,Z 280.57,A -85,B 0,C 180,E1 -554.897,E2 -554.897} C_VEL
LIN {X 0,Y 601.425,Z 280.569,A -85,B 0,C 180,E1 -556.986,E2 -556.986} C_VEL
LIN {X 0,Y 601.392,Z 280.566,A -85,B 0,C 180,E1 -559.81,E2 -559.81} C_VEL
LIN {X 0,Y 601.402,Z 280.564,A -85,B 0,C 180,E1 -561.959,E2 -561.959} C_VEL
LIN {X 0,Y 601.398,Z 280.573,A -85,B 0,C 180,E1 -564.879,E2 -564.879} C_VEL
LIN {X 0,Y 601.401,Z 280.572,A -85,B 0,C 180,E1 -567.359,E2 -567.359} C_VEL
LIN {X 0,Y 601.405,Z 280.573,A -85,B 0,C 180,E1 -569.394,E2 -569.394} C_VEL
LIN {X 0,Y 601.392,Z 280.57,A -85,B 0,C 180,E1 -571.727,E2 -571.727} C_VEL
LIN {X 0,Y 601.416,Z 280.564,A -85,B 0,C 180,E1 -574.119,E2 -574.119} C_VEL
LIN {X 0,Y 601.4,Z 280.565,A -85,B 0,C 180,E1 -576.583,E2 -576.583} C_VEL
LIN {X 0,Y 601.44,Z 280.57,A -85,B 0,C 180,E1 -579.535,E2 -579.535} C_VEL
LIN {X 0,Y 601.416,Z 280.574,A -85,B 0,C 180,E1 -581.766,E2 -581.766} C_VEL
LIN {X 0,Y 601.399,Z 280.566,A -85,B 0,C 180,E1 -584.532,E2 -584.532} C_VEL
LIN {X 0,Y 601.411,Z 280.566,A -85,B 0,C 180,E1 -587.409,E2 -587.409} C_VEL
LIN {X 0,Y 601.4,Z 280.576,A -85,B 0,C 180,E1 -590.004,E2 -590.004} C_VEL
LIN {X 0,Y 601.4,Z 280.568,A -85,B 0,C 180,E1 -592.622,E2 -592.622} C_VEL
LIN {X 0,Y 601.388,Z 280.566,A -85,B 0,C 180,E1 -595.066,E2 -595.066} C_VEL
LIN {X 0,Y 601.422,Z 280.562,A -85,B 0,C 180,E1 -597.483,E2 -597.483} C_VEL
LIN {X 0,Y 601.431,Z 280.563,A -85,B 0,C 180,E1 -599.851,E2 -599.851} C_VEL
LIN {X 0,Y 601.415,Z 280.568,A -85,B 0,C 180,E1 -602.887,E2 -602.887} C_VEL
LIN {X 0,Y 601.389,Z 280.569,A -85,B 0,C 180,E1 -605.12,E2 -605.12} C_VEL
LIN {X 0,Y 601.397,Z 280.566,A -85,B 0,C 180,E1 -608.04,E2 -608.04} C_VEL
LIN {X 0,Y 601.413,Z 280.574,A -85,B 0,C 180,E1 -610.9,E2 -610.9} C_VEL
LIN {X 0,Y 601.416,Z 280.563,A -85,B 0,C 180,E1 -613.712,E2 -613.712} C_VEL
LIN {X 0,Y 601.407,Z 280.566,A -85,B 0,C 180,E1 -616.483,E2 -616.483} C_VEL
LIN {X 0,Y 601.411,Z 280.574,A -85,B 0,C 180,E1 -619.223,E2 -619.223} C_VEL
LIN {X 0,Y 601.398,Z 280.567,A -85,B 0,C 180,E1 -621.938,E2 -621.938} C_VEL
LIN {X 0,Y 601.421,Z 280.631,A -85,B 0,C 180,E1 -624.635,E2 -624.635} C_VEL
LIN {X 0,Y 601.477,Z 295.606,A -85,B 0,C 180,E1 -627.153,E2 -627.153} C_VEL
LIN {X 0,Y 601.447,Z 312.794,A -85,B 0,C 180,E1 -629.999,E2 -629.999} C_VEL
LIN {X 0,Y 601.439,Z 318.146,A -85,B 0,C 180,E1 -630.878,E2 -630.878} C_VEL
LIN {X 0,Y 601.696,Z 322.234,A -85,B 0,C 180,E1 -630.941,E2 -630.941} C_VEL
LIN {X 0,Y 601.592,Z 425.593,A -85,B 0,C 180,E1 -632.196,E2 -632.196} C_VEL
LIN {X 0,Y 601.552,Z 439.211,A -85,B 0,C 180,E1 -632.51,E2 -632.51} C_VEL
LIN {X 0,Y 601.559,Z 451.445,A -85,B 0,C 180,E1 -632.929,E2 -632.929} C_VEL
LIN {X 0,Y 601.501,Z 462.475,A -85,B 0,C 180,E1 -633.432,E2 -633.432} C_VEL
LIN {X 0,Y 601.5,Z 473.931,A -85,B 0,C 180,E1 -634.103,E2 -634.103} C_VEL
LIN {X 0,Y 601.443,Z 484.213,A -85,B 0,C 180,E1 -634.859,E2 -634.859} C_VEL
LIN {X 0,Y 601.423,Z 491.871,A -85,B 0,C 180,E1 -635.532,E2 -635.532} C_VEL
LIN {X 0,Y 601.394,Z 500.203,A -85,B 0,C 180,E1 -636.404,E2 -636.404} C_VEL
LIN {X 0,Y 601.378,Z 507.836,A -85,B 0,C 180,E1 -637.385,E2 -637.385} C_VEL
LIN {X 0,Y 601.368,Z 514.165,A -85,B 0,C 180,E1 -638.399,E2 -638.399} C_VEL
LIN {X 0,Y 601.346,Z 519.221,A -85,B 0,C 180,E1 -639.416,E2 -639.416} C_VEL
LIN {X 0,Y 601.358,Z 523.139,A -85,B 0,C 180,E1 -640.436,E2 -640.436} C_VEL
LIN {X 0,Y 601.323,Z 526.025,A -85,B 0,C 180,E1 -641.46,E2 -641.46} C_VEL
LIN {X 0,Y 601.341,Z 527.379,A -85,B 0,C 180,E1 -642.143,E2 -642.143} C_VEL
LIN {X 0,Y 601.325,Z 528.328,A -85,B 0,C 180,E1 -642.83,E2 -642.83} C_VEL
LIN {X 0,Y 601.347,Z 528.999,A -85,B 0,C 180,E1 -644.063,E2 -644.063} C_VEL
LIN {X 0,Y 601.314,Z 528.656,A -85,B 0,C 180,E1 -644.899,E2 -644.899} C_VEL
LIN {X 0,Y 601.324,Z 527.94,A -85,B 0,C 180,E1 -645.593,E2 -645.593} C_VEL
LIN {X 0,Y 601.324,Z 526.114,A -85,B 0,C 180,E1 -646.589,E2 -646.589} C_VEL
LIN {X 0,Y 601.326,Z 523.027,A -85,B 0,C 180,E1 -647.69,E2 -647.69} C_VEL
LIN {X 0,Y 601.349,Z 518.675,A -85,B 0,C 180,E1 -648.8,E2 -648.8} C_VEL
LIN {X 0,Y 601.368,Z 512.434,A -85,B 0,C 180,E1 -649.988,E2 -649.988} C_VEL
LIN {X 0,Y 601.395,Z 504.99,A -85,B 0,C 180,E1 -651.094,E2 -651.094} C_VEL
LIN {X 0,Y 601.387,Z 497.797,A -85,B 0,C 180,E1 -651.959,E2 -651.959} C_VEL
LIN {X 0,Y 601.437,Z 488.616,A -85,B 0,C 180,E1 -652.863,E2 -652.863} C_VEL
LIN {X 0,Y 601.458,Z 478.385,A -85,B 0,C 180,E1 -653.682,E2 -653.682} C_VEL
LIN {X 0,Y 601.481,Z 467.525,A -85,B 0,C 180,E1 -654.383,E2 -654.383} C_VEL
LIN {X 0,Y 601.536,Z 454.998,A -85,B 0,C 180,E1 -655.01,E2 -655.01} C_VEL
LIN {X 0,Y 601.57,Z 442.769,A -85,B 0,C 180,E1 -655.471,E2 -655.471} C_VEL
LIN {X 0,Y 601.584,Z 429.993,A -85,B 0,C 180,E1 -655.811,E2 -655.811} C_VEL
LIN {X 0,Y 601.612,Z 415.85,A -85,B 0,C 180,E1 -656.03,E2 -656.03} C_VEL
LIN {X 0,Y 601.559,Z 319.145,A -85,B 0,C 180,E1 -657.19,E2 -657.19} C_VEL
LIN {X 0,Y 601.443,Z 318.061,A -85,B 0,C 180,E1 -657.226,E2 -657.226} C_VEL
LIN {X 0,Y 601.461,Z 301.471,A -85,B 0,C 180,E1 -659.962,E2 -659.962} C_VEL
LIN {X 0,Y 601.523,Z 284.899,A -85,B 0,C 180,E1 -662.731,E2 -662.731} C_VEL
LIN {X 0,Y 601.389,Z 280.57,A -85,B 0,C 180,E1 -663.489,E2 -663.489} C_VEL
LIN {X 0,Y 601.388,Z 280.569,A -85,B 0,C 180,E1 -666.259,E2 -666.259} C_VEL
LIN {X 0,Y 601.405,Z 280.569,A -85,B 0,C 180,E1 -668.468,E2 -668.468} C_VEL
LIN {X 0,Y 601.402,Z 280.575,A -85,B 0,C 180,E1 -670.874,E2 -670.874} C_VEL
LIN {X 0,Y 601.396,Z 280.568,A -85,B 0,C 180,E1 -673.588,E2 -673.588} C_VEL
LIN {X 0,Y 601.4,Z 280.566,A -85,B 0,C 180,E1 -676.429,E2 -676.429} C_VEL
LIN {X 0,Y 601.397,Z 280.573,A -85,B 0,C 180,E1 -679.427,E2 -679.427} C_VEL
LIN {X 0,Y 601.382,Z 280.571,A -85,B 0,C 180,E1 -681.729,E2 -681.729} C_VEL
LIN {X 0,Y 601.363,Z 280.57,A -85,B 0,C 180,E1 -684.244,E2 -684.244} C_VEL
LIN {X 0,Y 601.384,Z 280.567,A -85,B 0,C 180,E1 -686.684,E2 -686.684} C_VEL
LIN {X 0,Y 601.383,Z 280.571,A -85,B 0,C 180,E1 -689.056,E2 -689.056} C_VEL
LIN {X 0,Y 601.429,Z 280.569,A -85,B 0,C 180,E1 -691.373,E2 -691.373} C_VEL
LIN {X 0,Y 601.364,Z 280.57,A -85,B 0,C 180,E1 -694.38,E2 -694.38} C_VEL
LIN {X 0,Y 601.354,Z 280.571,A -85,B 0,C 180,E1 -696.587,E2 -696.587} C_VEL
LIN {X 0,Y 601.409,Z 280.569,A -85,B 0,C 180,E1 -699.478,E2 -699.478} C_VEL
LIN {X 0,Y 601.357,Z 280.574,A -85,B 0,C 180,E1 -702.311,E2 -702.311} C_VEL
LIN {X 0,Y 601.371,Z 280.572,A -85,B 0,C 180,E1 -704.408,E2 -704.408} C_VEL
LIN {X 0,Y 601.376,Z 280.571,A -85,B 0,C 180,E1 -706.483,E2 -706.483} C_VEL
LIN {X 0,Y 601.359,Z 280.57,A -85,B 0,C 180,E1 -709.015,E2 -709.015} C_VEL
LIN {X 0,Y 601.355,Z 280.57,A -85,B 0,C 180,E1 -711.261,E2 -711.261} C_VEL
LIN {X 0,Y 601.382,Z 280.573,A -85,B 0,C 180,E1 -713.963,E2 -713.963} C_VEL
LIN {X 0,Y 601.366,Z 280.574,A -85,B 0,C 180,E1 -716.65,E2 -716.65} C_VEL
LIN {X 0,Y 601.342,Z 280.572,A -85,B 0,C 180,E1 -719.331,E2 -719.331} C_VEL
LIN {X 0,Y 601.358,Z 280.57,A -85,B 0,C 180,E1 -721.339,E2 -721.339} C_VEL
LIN {X 0,Y 601.341,Z 280.573,A -85,B 0,C 180,E1 -723.35,E2 -723.35} C_VEL
LIN {X 0,Y 601.372,Z 280.569,A -85,B 0,C 180,E1 -725.365,E2 -725.365} C_VEL
LIN {X 0,Y 601.358,Z 280.571,A -85,B 0,C 180,E1 -727.386,E2 -727.386} C_VEL
LIN {X 0,Y 601.373,Z 280.569,A -85,B 0,C 180,E1 -729.417,E2 -729.417} C_VEL
LIN {X 0,Y 601.39,Z 280.567,A -85,B 0,C 180,E1 -731.459,E2 -731.459} C_VEL
LIN {X 0,Y 601.368,Z 280.57,A -85,B 0,C 180,E1 -734.207,E2 -734.207} C_VEL
LIN {X 0,Y 601.396,Z 280.576,A -85,B 0,C 180,E1 -736.987,E2 -736.987} C_VEL
LIN {X 0,Y 601.374,Z 280.569,A -85,B 0,C 180,E1 -739.811,E2 -739.811} C_VEL
LIN {X 0,Y 601.393,Z 280.569,A -85,B 0,C 180,E1 -742.684,E2 -742.684} C_VEL
LIN {X 0,Y 601.423,Z 280.566,A -85,B 0,C 180,E1 -745.618,E2 -745.618} C_VEL
LIN {X 0,Y 601.376,Z 280.57,A -85,B 0,C 180,E1 -747.87,E2 -747.87} C_VEL
LIN {X 0,Y 601.392,Z 280.566,A -85,B 0,C 180,E1 -750.166,E2 -750.166} C_VEL
LIN {X 0,Y 601.387,Z 280.567,A -85,B 0,C 180,E1 -752.712,E2 -752.712} C_VEL
LIN {X 0,Y 601.37,Z 280.573,A -85,B 0,C 180,E1 -755.11,E2 -755.11} C_VEL
LIN {X 0,Y 601.423,Z 280.571,A -85,B 0,C 180,E1 -757.42,E2 -757.42} C_VEL
LIN {X 0,Y 601.395,Z 280.571,A -85,B 0,C 180,E1 -759.997,E2 -759.997} C_VEL
LIN {X 0,Y 601.369,Z 280.568,A -85,B 0,C 180,E1 -762.674,E2 -762.674} C_VEL
LIN {X 0,Y 601.392,Z 280.567,A -85,B 0,C 180,E1 -764.533,E2 -764.533} C_VEL
LIN {X 0,Y 601.423,Z 280.564,A -85,B 0,C 180,E1 -766.428,E2 -766.428} C_VEL
LIN {X 0,Y 601.395,Z 280.566,A -85,B 0,C 180,E1 -769.125,E2 -769.125} C_VEL
LIN {X 0,Y 601.406,Z 280.571,A -85,B 0,C 180,E1 -771.732,E2 -771.732} C_VEL
LIN {X 0,Y 601.384,Z 280.575,A -85,B 0,C 180,E1 -774.246,E2 -774.246} C_VEL
LIN {X 0,Y 601.422,Z 280.565,A -85,B 0,C 180,E1 -776.687,E2 -776.687} C_VEL
LIN {X 0,Y 601.414,Z 280.564,A -85,B 0,C 180,E1 -779.059,E2 -779.059} C_VEL
LIN {X 0,Y 601.405,Z 280.565,A -85,B 0,C 180,E1 -781.373,E2 -781.373} C_VEL
LIN {X 0,Y 601.392,Z 280.567,A -85,B 0,C 180,E1 -783.637,E2 -783.637} C_VEL
LIN {X 0,Y 601.413,Z 280.574,A -85,B 0,C 180,E1 -786.59,E2 -786.59} C_VEL
LIN {X 0,Y 601.412,Z 280.604,A -85,B 0,C 180,E1 -787.556,E2 -787.556} C_VEL
LIN {X 0,Y 601.626,Z 289.026,A -85,B 0,C 180,E1 -788.77,E2 -788.77} C_VEL
LIN {X 0,Y 601.532,Z 307.496,A -85,B 0,C 180,E1 -791.377,E2 -791.377} C_VEL
LIN {X 0,Y 601.507,Z 326.806,A -85,B 0,C 180,E1 -794.064,E2 -794.064} C_VEL
LIN {X 0,Y 601.445,Z 346.798,A -85,B 0,C 180,E1 -796.808,E2 -796.808} C_VEL
LIN {X 0,Y 601.668,Z 352.568,A -85,B 0,C 180,E1 -796.899,E2 -796.899} C_VEL
LIN {X 0,Y 601.611,Z 454.984,A -85,B 0,C 180,E1 -798.14,E2 -798.14} C_VEL
LIN {X 0,Y 601.586,Z 468.242,A -85,B 0,C 180,E1 -798.439,E2 -798.439} C_VEL
LIN {X 0,Y 601.544,Z 479.981,A -85,B 0,C 180,E1 -798.828,E2 -798.828} C_VEL
LIN {X 0,Y 601.528,Z 490.938,A -85,B 0,C 180,E1 -799.312,E2 -799.312} C_VEL
LIN {X 0,Y 601.457,Z 501.592,A -85,B 0,C 180,E1 -799.906,E2 -799.906} C_VEL
LIN {X 0,Y 601.445,Z 512.484,A -85,B 0,C 180,E1 -800.67,E2 -800.67} C_VEL
LIN {X 0,Y 601.423,Z 521.323,A -85,B 0,C 180,E1 -801.432,E2 -801.432} C_VEL
LIN {X 0,Y 601.396,Z 529.483,A -85,B 0,C 180,E1 -802.277,E2 -802.277} C_VEL
LIN {X 0,Y 601.381,Z 537.475,A -85,B 0,C 180,E1 -803.289,E2 -803.289} C_VEL
LIN {X 0,Y 601.371,Z 543.87,A -85,B 0,C 180,E1 -804.3,E2 -804.3} C_VEL
LIN {X 0,Y 601.336,Z 548.953,A -85,B 0,C 180,E1 -805.308,E2 -805.308} C_VEL
LIN {X 0,Y 601.367,Z 552.898,A -85,B 0,C 180,E1 -806.315,E2 -806.315} C_VEL
LIN {X 0,Y 601.325,Z 555.81,A -85,B 0,C 180,E1 -807.321,E2 -807.321} C_VEL
LIN {X 0,Y 601.34,Z 557.203,A -85,B 0,C 180,E1 -807.991,E2 -807.991} C_VEL
LIN {X 0,Y 601.339,Z 558.784,A -85,B 0,C 180,E1 -809.331,E2 -809.331} C_VEL
LIN {X 0,Y 601.335,Z 559,A -85,B 0,C 180,E1 -810.001,E2 -810.001} C_VEL
LIN {X 0,Y 601.348,Z 558.184,A -85,B 0,C 180,E1 -811.34,E2 -811.34} C_VEL
LIN {X 0,Y 601.34,Z 557.201,A -85,B 0,C 180,E1 -812.01,E2 -812.01} C_VEL
LIN {X 0,Y 601.325,Z 555.808,A -85,B 0,C 180,E1 -812.68,E2 -812.68} C_VEL
LIN {X 0,Y 601.367,Z 552.894,A -85,B 0,C 180,E1 -813.686,E2 -813.686} C_VEL
LIN {X 0,Y 601.336,Z 548.947,A -85,B 0,C 180,E1 -814.693,E2 -814.693} C_VEL
LIN {X 0,Y 601.372,Z 542.874,A -85,B 0,C 180,E1 -815.87,E2 -815.87} C_VEL
LIN {X 0,Y 601.381,Z 536.231,A -85,B 0,C 180,E1 -816.88,E2 -816.88} C_VEL
LIN {X 0,Y 601.4,Z 527.984,A -85,B 0,C 180,E1 -817.893,E2 -817.893} C_VEL
LIN {X 0,Y 601.433,Z 519.531,A -85,B 0,C 180,E1 -818.738,E2 -818.738} C_VEL
LIN {X 0,Y 601.44,Z 509.085,A -85,B 0,C 180,E1 -819.586,E2 -819.586} C_VEL
LIN {X 0,Y 601.472,Z 498.749,A -85,B 0,C 180,E1 -820.265,E2 -820.265} C_VEL
LIN {X 0,Y 601.54,Z 486.574,A -85,B 0,C 180,E1 -820.897,E2 -820.897} C_VEL
LIN {X 0,Y 601.569,Z 474.199,A -85,B 0,C 180,E1 -821.379,E2 -821.379} C_VEL
LIN {X 0,Y 601.586,Z 461.415,A -85,B 0,C 180,E1 -821.733,E2 -821.733} C_VEL
LIN {X 0,Y 601.616,Z 449.043,A -85,B 0,C 180,E1 -821.946,E2 -821.946} C_VEL
LIN {X 0,Y 601.553,Z 347.769,A -85,B 0,C 180,E1 -823.161,E2 -823.161} C_VEL
LIN {X 0,Y 601.445,Z 346.788,A -85,B 0,C 180,E1 -823.193,E2 -823.193} C_VEL
LIN {X 0,Y 601.507,Z 326.797,A -85,B 0,C 180,E1 -825.937,E2 -825.937} C_VEL
LIN {X 0,Y 601.532,Z 307.493,A -85,B 0,C 180,E1 -828.623,E2 -828.623} C_VEL
LIN {X 0,Y 601.656,Z 287.758,A -85,B 0,C 180,E1 -831.41,E2 -831.41} C_VEL
LIN {X 0,Y 601.411,Z 280.568,A -85,B 0,C 180,E1 -832.469,E2 -832.469} C_VEL
LIN {X 0,Y 601.4,Z 280.566,A -85,B 0,C 180,E1 -834.879,E2 -834.879} C_VEL
LIN {X 0,Y 601.421,Z 280.568,A -85,B 0,C 180,E1 -837.363,E2 -837.363} C_VEL
LIN {X 0,Y 601.406,Z 280.569,A -85,B 0,C 180,E1 -840.166,E2 -840.166} C_VEL
LIN {X 0,Y 601.406,Z 280.564,A -85,B 0,C 180,E1 -842.713,E2 -842.713} C_VEL
LIN {X 0,Y 601.383,Z 280.567,A -85,B 0,C 180,E1 -845.11,E2 -845.11} C_VEL
LIN {X 0,Y 601.435,Z 280.561,A -85,B 0,C 180,E1 -847.419,E2 -847.419} C_VEL
LIN {X 0,Y 601.403,Z 280.572,A -85,B 0,C 180,E1 -849.996,E2 -849.996} C_VEL
LIN {X 0,Y 601.387,Z 280.571,A -85,B 0,C 180,E1 -852.673,E2 -852.673} C_VEL
LIN {X 0,Y 601.402,Z 280.564,A -85,B 0,C 180,E1 -855.479,E2 -855.479} C_VEL
LIN {X 0,Y 601.425,Z 280.571,A -85,B 0,C 180,E1 -858.407,E2 -858.407} C_VEL
LIN {X 0,Y 601.399,Z 280.571,A -85,B 0,C 180,E1 -860.872,E2 -860.872} C_VEL
LIN {X 0,Y 601.391,Z 280.567,A -85,B 0,C 180,E1 -863.416,E2 -863.416} C_VEL
LIN {X 0,Y 601.432,Z 280.561,A -85,B 0,C 180,E1 -866.065,E2 -866.065} C_VEL
LIN {X 0,Y 601.403,Z 280.573,A -85,B 0,C 180,E1 -869.057,E2 -869.057} C_VEL
LIN {X 0,Y 601.414,Z 280.568,A -85,B 0,C 180,E1 -871.372,E2 -871.372} C_VEL
LIN {X 0,Y 601.392,Z 280.568,A -85,B 0,C 180,E1 -873.636,E2 -873.636} C_VEL
LIN {X 0,Y 601.407,Z 280.565,A -85,B 0,C 180,E1 -875.857,E2 -875.857} C_VEL
LIN {X 0,Y 601.393,Z 280.566,A -85,B 0,C 180,E1 -878.04,E2 -878.04} C_VEL
LIN {X 0,Y 601.393,Z 280.566,A -85,B 0,C 180,E1 -880.19,E2 -880.19} C_VEL
LIN {X 0,Y 601.432,Z 280.564,A -85,B 0,C 180,E1 -883.014,E2 -883.014} C_VEL
LIN {X 0,Y 601.402,Z 280.57,A -85,B 0,C 180,E1 -885.917,E2 -885.917} C_VEL
LIN {X 0,Y 601.408,Z 280.564,A -85,B 0,C 180,E1 -888.541,E2 -888.541} C_VEL
LIN {X 0,Y 601.414,Z 280.566,A -85,B 0,C 180,E1 -891.262,E2 -891.262} C_VEL
LIN {X 0,Y 601.405,Z 280.574,A -85,B 0,C 180,E1 -893.963,E2 -893.963} C_VEL
LIN {X 0,Y 601.405,Z 280.576,A -85,B 0,C 180,E1 -895.979,E2 -895.979} C_VEL
LIN {X 0,Y 601.437,Z 280.571,A -85,B 0,C 180,E1 -897.991,E2 -897.991} C_VEL
LIN {X 0,Y 601.427,Z 280.564,A -85,B 0,C 180,E1 -900.669,E2 -900.669} C_VEL
LIN {X 0,Y 601.413,Z 280.563,A -85,B 0,C 180,E1 -903.349,E2 -903.349} C_VEL
LIN {X 0,Y 601.414,Z 280.569,A -85,B 0,C 180,E1 -906.037,E2 -906.037} C_VEL
LIN {X 0,Y 601.406,Z 280.57,A -85,B 0,C 180,E1 -908.738,E2 -908.738} C_VEL
LIN {X 0,Y 601.406,Z 280.567,A -85,B 0,C 180,E1 -911.001,E2 -911.001} C_VEL
LIN {X 0,Y 601.407,Z 280.568,A -85,B 0,C 180,E1 -912.363,E2 -912.363} C_VEL
LIN {X 0,Y 600.738,Z 280.655,A -85,B 0,C 180,E1 -912.923,E2 -912.923} C_VEL
LIN {X 0,Y 597.887,Z 281.01,A -85,B 0,C 180,E1 -913.83,E2 -913.83} C_VEL
LIN {X 0,Y 595.477,Z 281.312,A -85,B 0,C 180,E1 -914.561,E2 -914.561} C_VEL
LIN {X 0,Y 594.438,Z 281.436,A -85,B 0,C 180,E1 -915.124,E2 -915.124} C_VEL
LIN {X 0,Y 594.351,Z 281.445,A -85,B 0,C 180,E1 -915.315,E2 -915.315} C_VEL
LIN {X 0,Y 594.382,Z 281.443,A -85,B 0,C 180,E1 -917.193,E2 -917.193} C_VEL
LIN {X 0,Y 594.368,Z 281.441,A -85,B 0,C 180,E1 -920.054,E2 -920.054} C_VEL
LIN {X 0,Y 594.354,Z 281.454,A -85,B 0,C 180,E1 -922.968,E2 -922.968} C_VEL
LIN {X 0,Y 594.358,Z 281.451,A -85,B 0,C 180,E1 -925.194,E2 -925.194} C_VEL
LIN {X 0,Y 594.349,Z 281.448,A -85,B 0,C 180,E1 -927.519,E2 -927.519} C_VEL
LIN {X 0,Y 594.358,Z 281.445,A -85,B 0,C 180,E1 -929.777,E2 -929.777} C_VEL
LIN {X 0,Y 594.356,Z 281.443,A -85,B 0,C 180,E1 -932.148,E2 -932.148} C_VEL
LIN {X 0,Y 594.392,Z 281.438,A -85,B 0,C 180,E1 -934.579,E2 -934.579} C_VEL
LIN {X 0,Y 594.387,Z 281.449,A -85,B 0,C 180,E1 -937.608,E2 -937.608} C_VEL
LIN {X 0,Y 594.361,Z 281.442,A -85,B 0,C 180,E1 -940.567,E2 -940.567} C_VEL
LIN {X 0,Y 594.36,Z 281.445,A -85,B 0,C 180,E1 -943.3,E2 -943.3} C_VEL
LIN {X 0,Y 594.353,Z 281.449,A -85,B 0,C 180,E1 -946.162,E2 -946.162} C_VEL
LIN {X 0,Y 594.369,Z 281.443,A -85,B 0,C 180,E1 -948.535,E2 -948.535} C_VEL
LIN {X 0,Y 594.37,Z 281.441,A -85,B 0,C 180,E1 -951.297,E2 -951.297} C_VEL
LIN {X 0,Y 594.36,Z 281.446,A -85,B 0,C 180,E1 -953.756,E2 -953.756} C_VEL
LIN {X 0,Y 594.375,Z 281.451,A -85,B 0,C 180,E1 -956.238,E2 -956.238} C_VEL
LIN {X 0,Y 594.365,Z 281.447,A -85,B 0,C 180,E1 -958.649,E2 -958.649} C_VEL
LIN {X 0,Y 594.375,Z 281.442,A -85,B 0,C 180,E1 -961.043,E2 -961.043} C_VEL
LIN {X 0,Y 594.363,Z 281.442,A -85,B 0,C 180,E1 -963.299,E2 -963.299} C_VEL
LIN {X 0,Y 594.355,Z 281.442,A -85,B 0,C 180,E1 -965.573,E2 -965.573} C_VEL
LIN {X 0,Y 594.357,Z 281.449,A -85,B 0,C 180,E1 -968.496,E2 -968.496} C_VEL
LIN {X 0,Y 594.363,Z 281.444,A -85,B 0,C 180,E1 -971.381,E2 -971.381} C_VEL
LIN {X 0,Y 594.357,Z 281.443,A -85,B 0,C 180,E1 -974.218,E2 -974.218} C_VEL
LIN {X 0,Y 594.368,Z 281.442,A -85,B 0,C 180,E1 -976.32,E2 -976.32} C_VEL
LIN {X 0,Y 594.372,Z 281.451,A -85,B 0,C 180,E1 -979.094,E2 -979.094} C_VEL
LIN {X 0,Y 594.353,Z 281.445,A -85,B 0,C 180,E1 -981.842,E2 -981.842} C_VEL
LIN {X 0,Y 594.403,Z 281.528,A -85,B 0,C 180,E1 -984.55,E2 -984.55} C_VEL
LIN {X 0,Y 594.484,Z 294.613,A -85,B 0,C 180,E1 -986.78,E2 -986.78} C_VEL
LIN {X 0,Y 594.408,Z 311.781,A -85,B 0,C 180,E1 -989.661,E2 -989.661} C_VEL
LIN {X 0,Y 594.398,Z 318.145,A -85,B 0,C 180,E1 -990.719,E2 -990.719} C_VEL
LIN {X 0,Y 594.777,Z 323.718,A -85,B 0,C 180,E1 -990.803,E2 -990.803} C_VEL
LIN {X 0,Y 594.671,Z 425.386,A -85,B 0,C 180,E1 -992.052,E2 -992.052} C_VEL
LIN {X 0,Y 594.581,Z 438.364,A -85,B 0,C 180,E1 -992.349,E2 -992.349} C_VEL
LIN {X 0,Y 594.574,Z 451.373,A -85,B 0,C 180,E1 -992.794,E2 -992.794} C_VEL
LIN {X 0,Y 594.51,Z 462.419,A -85,B 0,C 180,E1 -993.303,E2 -993.303} C_VEL
LIN {X 0,Y 594.471,Z 473.897,A -85,B 0,C 180,E1 -993.982,E2 -993.982} C_VEL
LIN {X 0,Y 594.419,Z 484.195,A -85,B 0,C 180,E1 -994.747,E2 -994.747} C_VEL
LIN {X 0,Y 594.384,Z 491.856,A -85,B 0,C 180,E1 -995.427,E2 -995.427} C_VEL
LIN {X 0,Y 594.328,Z 501.037,A -85,B 0,C 180,E1 -996.409,E2 -996.409} C_VEL
LIN {X 0,Y 594.293,Z 508.947,A -85,B 0,C 180,E1 -997.474,E2 -997.474} C_VEL
LIN {X 0,Y 594.298,Z 515.06,A -85,B 0,C 180,E1 -998.5,E2 -998.5} C_VEL
LIN {X 0,Y 594.268,Z 519.925,A -85,B 0,C 180,E1 -999.53,E2 -999.53} C_VEL
LIN {X 0,Y 594.282,Z 523.665,A -85,B 0,C 180,E1 -1000.562,E2 -1000.562} C_VEL
LIN {X 0,Y 594.232,Z 526.384,A -85,B 0,C 180,E1 -1001.598,E2 -1001.598} C_VEL
LIN {X 0,Y 594.238,Z 527.655,A -85,B 0,C 180,E1 -1002.291,E2 -1002.291} C_VEL
LIN {X 0,Y 594.243,Z 528.516,A -85,B 0,C 180,E1 -1002.985,E2 -1002.985} C_VEL
LIN {X 0,Y 594.258,Z 528.988,A -85,B 0,C 180,E1 -1004.124,E2 -1004.124} C_VEL
LIN {X 0,Y 594.209,Z 528.535,A -85,B 0,C 180,E1 -1005.081,E2 -1005.081} C_VEL
LIN {X 0,Y 594.251,Z 527.68,A -85,B 0,C 180,E1 -1005.783,E2 -1005.783} C_VEL
LIN {X 0,Y 594.238,Z 526.007,A -85,B 0,C 180,E1 -1006.669,E2 -1006.669} C_VEL
LIN {X 0,Y 594.24,Z 522.428,A -85,B 0,C 180,E1 -1007.908,E2 -1007.908} C_VEL
LIN {X 0,Y 594.279,Z 517.631,A -85,B 0,C 180,E1 -1009.077,E2 -1009.077} C_VEL
LIN {X 0,Y 594.297,Z 511.384,A -85,B 0,C 180,E1 -1010.236,E2 -1010.236} C_VEL
LIN {X 0,Y 594.315,Z 505.078,A -85,B 0,C 180,E1 -1011.167,E2 -1011.167} C_VEL
LIN {X 0,Y 594.344,Z 497.825,A -85,B 0,C 180,E1 -1012.051,E2 -1012.051} C_VEL
LIN {X 0,Y 594.407,Z 487.584,A -85,B 0,C 180,E1 -1013.057,E2 -1013.057} C_VEL
LIN {X 0,Y 594.448,Z 477.168,A -85,B 0,C 180,E1 -1013.886,E2 -1013.886} C_VEL
LIN {X 0,Y 594.487,Z 465.993,A -85,B 0,C 180,E1 -1014.592,E2 -1014.592} C_VEL
LIN {X 0,Y 594.565,Z 454.014,A -85,B 0,C 180,E1 -1015.184,E2 -1015.184} C_VEL
LIN {X 0,Y 594.584,Z 441.442,A -85,B 0,C 180,E1 -1015.651,E2 -1015.651} C_VEL
LIN {X 0,Y 594.622,Z 428.258,A -85,B 0,C 180,E1 -1015.984,E2 -1015.984} C_VEL
LIN {X 0,Y 594.671,Z 409.834,A -85,B 0,C 180,E1 -1016.245,E2 -1016.245} C_VEL
LIN {X 0,Y 594.741,Z 320.449,A -85,B 0,C 180,E1 -1017.327,E2 -1017.327} C_VEL
LIN {X 0,Y 594.387,Z 318.188,A -85,B 0,C 180,E1 -1017.364,E2 -1017.364} C_VEL
LIN {X 0,Y 594.451,Z 302.06,A -85,B 0,C 180,E1 -1020.055,E2 -1020.055} C_VEL
LIN {X 0,Y 594.503,Z 285.006,A -85,B 0,C 180,E1 -1022.941,E2 -1022.941} C_VEL
LIN {X 0,Y 594.352,Z 281.447,A -85,B 0,C 180,E1 -1023.558,E2 -1023.558} C_VEL
LIN {X 0,Y 594.361,Z 281.448,A -85,B 0,C 180,E1 -1026.48,E2 -1026.48} C_VEL
LIN {X 0,Y 594.361,Z 281.452,A -85,B 0,C 180,E1 -1028.806,E2 -1028.806} C_VEL
LIN {X 0,Y 594.358,Z 281.443,A -85,B 0,C 180,E1 -1031.846,E2 -1031.846} C_VEL
LIN {X 0,Y 594.329,Z 281.452,A -85,B 0,C 180,E1 -1034.805,E2 -1034.805} C_VEL
LIN {X 0,Y 594.336,Z 281.448,A -85,B 0,C 180,E1 -1037.622,E2 -1037.622} C_VEL
LIN {X 0,Y 594.345,Z 281.444,A -85,B 0,C 180,E1 -1040.317,E2 -1040.317} C_VEL
LIN {X 0,Y 594.371,Z 281.445,A -85,B 0,C 180,E1 -1042.912,E2 -1042.912} C_VEL
LIN {X 0,Y 594.358,Z 281.445,A -85,B 0,C 180,E1 -1045.863,E2 -1045.863} C_VEL
LIN {X 0,Y 594.346,Z 281.444,A -85,B 0,C 180,E1 -1048.648,E2 -1048.648} C_VEL
LIN {X 0,Y 594.369,Z 281.443,A -85,B 0,C 180,E1 -1051.043,E2 -1051.043} C_VEL
LIN {X 0,Y 594.328,Z 281.45,A -85,B 0,C 180,E1 -1054.054,E2 -1054.054} C_VEL
LIN {X 0,Y 594.346,Z 281.446,A -85,B 0,C 180,E1 -1056.294,E2 -1056.294} C_VEL
LIN {X 0,Y 594.379,Z 281.441,A -85,B 0,C 180,E1 -1059.224,E2 -1059.224} C_VEL
LIN {X 0,Y 594.314,Z 281.455,A -85,B 0,C 180,E1 -1062.094,E2 -1062.094} C_VEL
LIN {X 0,Y 594.327,Z 281.453,A -85,B 0,C 180,E1 -1064.218,E2 -1064.218} C_VEL
LIN {X 0,Y 594.35,Z 281.449,A -85,B 0,C 180,E1 -1066.32,E2 -1066.32} C_VEL
LIN {X 0,Y 594.305,Z 281.449,A -85,B 0,C 180,E1 -1069.094,E2 -1069.094} C_VEL
LIN {X 0,Y 594.356,Z 281.447,A -85,B 0,C 180,E1 -1071.843,E2 -1071.843} C_VEL
LIN {X 0,Y 594.351,Z 281.449,A -85,B 0,C 180,E1 -1074.572,E2 -1074.572} C_VEL
LIN {X 0,Y 594.344,Z 281.443,A -85,B 0,C 180,E1 -1077.289,E2 -1077.289} C_VEL
LIN {X 0,Y 594.372,Z 281.444,A -85,B 0,C 180,E1 -1080,E2 -1080} C_VEL
LIN {X 0,Y 594.398,Z 281.445,A -85,B 0,C 180,E1 -1082.711,E2 -1082.711} C_VEL
LIN {X 0,Y 594.339,Z 281.445,A -85,B 0,C 180,E1 -1085.428,E2 -1085.428} C_VEL
LIN {X 0,Y 594.329,Z 281.445,A -85,B 0,C 180,E1 -1087.474,E2 -1087.474} C_VEL
LIN {X 0,Y 594.321,Z 281.447,A -85,B 0,C 180,E1 -1089.53,E2 -1089.53} C_VEL
LIN {X 0,Y 594.358,Z 281.442,A -85,B 0,C 180,E1 -1091.597,E2 -1091.597} C_VEL
LIN {X 0,Y 594.333,Z 281.448,A -85,B 0,C 180,E1 -1094.379,E2 -1094.379} C_VEL
LIN {X 0,Y 594.36,Z 281.448,A -85,B 0,C 180,E1 -1097.194,E2 -1097.194} C_VEL
LIN {X 0,Y 594.342,Z 281.444,A -85,B 0,C 180,E1 -1100.055,E2 -1100.055} C_VEL
LIN {X 0,Y 594.34,Z 281.452,A -85,B 0,C 180,E1 -1102.968,E2 -1102.968} C_VEL
LIN {X 0,Y 594.351,Z 281.444,A -85,B 0,C 180,E1 -1105.945,E2 -1105.945} C_VEL
LIN {X 0,Y 594.343,Z 281.444,A -85,B 0,C 180,E1 -1108.229,E2 -1108.229} C_VEL
LIN {X 0,Y 594.354,Z 281.443,A -85,B 0,C 180,E1 -1110.561,E2 -1110.561} C_VEL
LIN {X 0,Y 594.365,Z 281.444,A -85,B 0,C 180,E1 -1112.951,E2 -1112.951} C_VEL
LIN {X 0,Y 594.338,Z 281.454,A -85,B 0,C 180,E1 -1115.41,E2 -1115.41} C_VEL
LIN {X 0,Y 594.373,Z 281.445,A -85,B 0,C 180,E1 -1117.942,E2 -1117.942} C_VEL
LIN {X 0,Y 594.355,Z 281.443,A -85,B 0,C 180,E1 -1120.821,E2 -1120.821} C_VEL
LIN {X 0,Y 594.351,Z 281.446,A -85,B 0,C 180,E1 -1123.301,E2 -1123.301} C_VEL
LIN {X 0,Y 594.355,Z 281.448,A -85,B 0,C 180,E1 -1126.162,E2 -1126.162} C_VEL
LIN {X 0,Y 594.372,Z 281.443,A -85,B 0,C 180,E1 -1128.537,E2 -1128.537} C_VEL
LIN {X 0,Y 594.363,Z 281.443,A -85,B 0,C 180,E1 -1131.299,E2 -1131.299} C_VEL
LIN {X 0,Y 594.344,Z 281.45,A -85,B 0,C 180,E1 -1133.756,E2 -1133.756} C_VEL
LIN {X 0,Y 594.375,Z 281.45,A -85,B 0,C 180,E1 -1136.24,E2 -1136.24} C_VEL
LIN {X 0,Y 594.385,Z 281.443,A -85,B 0,C 180,E1 -1138.652,E2 -1138.652} C_VEL
LIN {X 0,Y 594.373,Z 281.441,A -85,B 0,C 180,E1 -1141.044,E2 -1141.044} C_VEL
LIN {X 0,Y 594.381,Z 281.44,A -85,B 0,C 180,E1 -1143.301,E2 -1143.301} C_VEL
LIN {X 0,Y 594.348,Z 281.446,A -85,B 0,C 180,E1 -1145.576,E2 -1145.576} C_VEL
LIN {X 0,Y 594.384,Z 281.542,A -85,B 0,C 180,E1 -1147.412,E2 -1147.412} C_VEL
LIN {X 0,Y 594.736,Z 287.767,A -85,B 0,C 180,E1 -1148.33,E2 -1148.33} C_VEL
LIN {X 0,Y 594.6,Z 307.305,A -85,B 0,C 180,E1 -1151.125,E2 -1151.125} C_VEL
LIN {X 0,Y 594.513,Z 325.547,A -85,B 0,C 180,E1 -1153.695,E2 -1153.695} C_VEL
LIN {X 0,Y 594.426,Z 345.696,A -85,B 0,C 180,E1 -1156.497,E2 -1156.497} C_VEL
LIN {X 0,Y 594.46,Z 347.202,A -85,B 0,C 180,E1 -1156.672,E2 -1156.672} C_VEL
LIN {X 0,Y 594.743,Z 354.357,A -85,B 0,C 180,E1 -1156.765,E2 -1156.765} C_VEL
LIN {X 0,Y 594.662,Z 454.984,A -85,B 0,C 180,E1 -1158,E2 -1158} C_VEL
LIN {X 0,Y 594.633,Z 468.243,A -85,B 0,C 180,E1 -1158.302,E2 -1158.302} C_VEL
LIN {X 0,Y 594.565,Z 480.43,A -85,B 0,C 180,E1 -1158.713,E2 -1158.713} C_VEL
LIN {X 0,Y 594.535,Z 492.645,A -85,B 0,C 180,E1 -1159.271,E2 -1159.271} C_VEL
LIN {X 0,Y 594.461,Z 504.211,A -85,B 0,C 180,E1 -1159.958,E2 -1159.958} C_VEL
LIN {X 0,Y 594.412,Z 514.532,A -85,B 0,C 180,E1 -1160.73,E2 -1160.73} C_VEL
LIN {X 0,Y 594.349,Z 523.036,A -85,B 0,C 180,E1 -1161.501,E2 -1161.501} C_VEL
LIN {X 0,Y 594.347,Z 530.966,A -85,B 0,C 180,E1 -1162.356,E2 -1162.356} C_VEL
LIN {X 0,Y 594.28,Z 538.83,A -85,B 0,C 180,E1 -1163.411,E2 -1163.411} C_VEL
LIN {X 0,Y 594.289,Z 545.684,A -85,B 0,C 180,E1 -1164.572,E2 -1164.572} C_VEL
LIN {X 0,Y 594.27,Z 550.374,A -85,B 0,C 180,E1 -1165.592,E2 -1165.592} C_VEL
LIN {X 0,Y 594.268,Z 553.958,A -85,B 0,C 180,E1 -1166.611,E2 -1166.611} C_VEL
LIN {X 0,Y 594.226,Z 555.81,A -85,B 0,C 180,E1 -1167.289,E2 -1167.289} C_VEL
LIN {X 0,Y 594.239,Z 557.202,A -85,B 0,C 180,E1 -1167.967,E2 -1167.967} C_VEL
LIN {X 0,Y 594.239,Z 558.784,A -85,B 0,C 180,E1 -1169.323,E2 -1169.323} C_VEL
LIN {X 0,Y 594.236,Z 559,A -85,B 0,C 180,E1 -1170.001,E2 -1170.001} C_VEL
LIN {X 0,Y 594.248,Z 558.184,A -85,B 0,C 180,E1 -1171.356,E2 -1171.356} C_VEL
LIN {X 0,Y 594.239,Z 557.201,A -85,B 0,C 180,E1 -1172.034,E2 -1172.034} C_VEL
LIN {X 0,Y 594.226,Z 555.808,A -85,B 0,C 180,E1 -1172.712,E2 -1172.712} C_VEL
LIN {X 0,Y 594.288,Z 552.894,A -85,B 0,C 180,E1 -1173.73,E2 -1173.73} C_VEL
LIN {X 0,Y 594.241,Z 548.947,A -85,B 0,C 180,E1 -1174.749,E2 -1174.749} C_VEL
LIN {X 0,Y 594.304,Z 542.874,A -85,B 0,C 180,E1 -1175.94,E2 -1175.94} C_VEL
LIN {X 0,Y 594.308,Z 536.232,A -85,B 0,C 180,E1 -1176.963,E2 -1176.963} C_VEL
LIN {X 0,Y 594.359,Z 527.985,A -85,B 0,C 180,E1 -1177.987,E2 -1177.987} C_VEL
LIN {X 0,Y 594.383,Z 519.531,A -85,B 0,C 180,E1 -1178.843,E2 -1178.843} C_VEL
LIN {X 0,Y 594.421,Z 509.087,A -85,B 0,C 180,E1 -1179.7,E2 -1179.7} C_VEL
LIN {X 0,Y 594.485,Z 498.75,A -85,B 0,C 180,E1 -1180.387,E2 -1180.387} C_VEL
LIN {X 0,Y 594.56,Z 487.698,A -85,B 0,C 180,E1 -1180.974,E2 -1180.974} C_VEL
LIN {X 0,Y 594.59,Z 475.69,A -85,B 0,C 180,E1 -1181.465,E2 -1181.465} C_VEL
LIN {X 0,Y 594.646,Z 462.328,A -85,B 0,C 180,E1 -1181.851,E2 -1181.851} C_VEL
LIN {X 0,Y 594.693,Z 449.043,A -85,B 0,C 180,E1 -1182.088,E2 -1182.088} C_VEL
LIN {X 0,Y 594.703,Z 348.887,A -85,B 0,C 180,E1 -1183.302,E2 -1183.302} C_VEL
LIN {X 0,Y 594.422,Z 346.788,A -85,B 0,C 180,E1 -1183.352,E2 -1183.352} C_VEL
LIN {X 0,Y 594.51,Z 326.797,A -85,B 0,C 180,E1 -1186.13,E2 -1186.13} C_VEL
LIN {X 0,Y 594.555,Z 309.166,A -85,B 0,C 180,E1 -1188.612,E2 -1188.612} C_VEL
LIN {X 0,Y 594.713,Z 290.077,A -85,B 0,C 180,E1 -1191.338,E2 -1191.338} C_VEL
LIN {X 0,Y 594.466,Z 282.023,A -85,B 0,C 180,E1 -1192.514,E2 -1192.514} C_VEL
LIN {X 0,Y 594.381,Z 281.445,A -85,B 0,C 180,E1 -1192.622,E2 -1192.622} C_VEL
LIN {X 0,Y 594.378,Z 281.444,A -85,B 0,C 180,E1 -1195.193,E2 -1195.193} C_VEL
LIN {X 0,Y 594.391,Z 281.446,A -85,B 0,C 180,E1 -1197.527,E2 -1197.527} C_VEL
LIN {X 0,Y 594.371,Z 281.443,A -85,B 0,C 180,E1 -1200.325,E2 -1200.325} C_VEL
LIN {X 0,Y 594.378,Z 281.439,A -85,B 0,C 180,E1 -1202.951,E2 -1202.951} C_VEL
LIN {X 0,Y 594.331,Z 281.447,A -85,B 0,C 180,E1 -1205.411,E2 -1205.411} C_VEL
LIN {X 0,Y 594.386,Z 281.447,A -85,B 0,C 180,E1 -1207.941,E2 -1207.941} C_VEL
LIN {X 0,Y 594.367,Z 281.443,A -85,B 0,C 180,E1 -1210.821,E2 -1210.821} C_VEL
LIN {X 0,Y 594.349,Z 281.443,A -85,B 0,C 180,E1 -1213.302,E2 -1213.302} C_VEL
LIN {X 0,Y 594.363,Z 281.448,A -85,B 0,C 180,E1 -1216.161,E2 -1216.161} C_VEL
LIN {X 0,Y 594.381,Z 281.451,A -85,B 0,C 180,E1 -1218.536,E2 -1218.536} C_VEL
LIN {X 0,Y 594.37,Z 281.442,A -85,B 0,C 180,E1 -1221.298,E2 -1221.298} C_VEL
LIN {X 0,Y 594.35,Z 281.443,A -85,B 0,C 180,E1 -1223.755,E2 -1223.755} C_VEL
LIN {X 0,Y 594.376,Z 281.442,A -85,B 0,C 180,E1 -1226.238,E2 -1226.238} C_VEL
LIN {X 0,Y 594.37,Z 281.447,A -85,B 0,C 180,E1 -1228.649,E2 -1228.649} C_VEL
LIN {X 0,Y 594.382,Z 281.45,A -85,B 0,C 180,E1 -1231.043,E2 -1231.043} C_VEL
LIN {X 0,Y 594.381,Z 281.446,A -85,B 0,C 180,E1 -1233.3,E2 -1233.3} C_VEL
LIN {X 0,Y 594.346,Z 281.448,A -85,B 0,C 180,E1 -1235.576,E2 -1235.576} C_VEL
LIN {X 0,Y 594.35,Z 281.446,A -85,B 0,C 180,E1 -1237.766,E2 -1237.766} C_VEL
LIN {X 0,Y 594.366,Z 281.443,A -85,B 0,C 180,E1 -1239.946,E2 -1239.946} C_VEL
LIN {X 0,Y 594.387,Z 281.44,A -85,B 0,C 180,E1 -1242.806,E2 -1242.806} C_VEL
LIN {X 0,Y 594.378,Z 281.446,A -85,B 0,C 180,E1 -1245.832,E2 -1245.832} C_VEL
LIN {X 0,Y 594.377,Z 281.44,A -85,B 0,C 180,E1 -1248.404,E2 -1248.404} C_VEL
LIN {X 0,Y 594.378,Z 281.441,A -85,B 0,C 180,E1 -1251.158,E2 -1251.158} C_VEL
LIN {X 0,Y 594.361,Z 281.453,A -85,B 0,C 180,E1 -1253.891,E2 -1253.891} C_VEL
LIN {X 0,Y 594.359,Z 281.453,A -85,B 0,C 180,E1 -1255.931,E2 -1255.931} C_VEL
LIN {X 0,Y 594.407,Z 281.447,A -85,B 0,C 180,E1 -1257.967,E2 -1257.967} C_VEL
LIN {X 0,Y 594.401,Z 281.439,A -85,B 0,C 180,E1 -1260.677,E2 -1260.677} C_VEL
LIN {X 0,Y 594.365,Z 281.441,A -85,B 0,C 180,E1 -1263.389,E2 -1263.389} C_VEL
LIN {X 0,Y 594.364,Z 281.448,A -85,B 0,C 180,E1 -1266.109,E2 -1266.109} C_VEL
LIN {X 0,Y 594.372,Z 281.445,A -85,B 0,C 180,E1 -1268.842,E2 -1268.842} C_VEL
LIN {X 0,Y 594.377,Z 281.439,A -85,B 0,C 180,E1 -1271.596,E2 -1271.596} C_VEL
LIN {X 0,Y 594.391,Z 281.444,A -85,B 0,C 180,E1 -1274.377,E2 -1274.377} C_VEL
LIN {X 0,Y 594.351,Z 281.445,A -85,B 0,C 180,E1 -1275.315,E2 -1275.315} C_VEL
LIN {X 0,Y 593.673,Z 281.53,A -85,B 0,C 180,E1 -1275.881,E2 -1275.881} C_VEL
LIN {X 0,Y 590.801,Z 281.896,A -85,B 0,C 180,E1 -1276.799,E2 -1276.799} C_VEL
LIN {X 0,Y 588.391,Z 282.19,A -85,B 0,C 180,E1 -1277.538,E2 -1277.538} C_VEL
LIN {X 0,Y 587.372,Z 282.314,A -85,B 0,C 180,E1 -1278.108,E2 -1278.108} C_VEL
LIN {X 0,Y 587.298,Z 282.324,A -85,B 0,C 180,E1 -1278.301,E2 -1278.301} C_VEL
LIN {X 0,Y 587.334,Z 282.326,A -85,B 0,C 180,E1 -1281.037,E2 -1281.037} C_VEL
LIN {X 0,Y 587.309,Z 282.327,A -85,B 0,C 180,E1 -1283.259,E2 -1283.259} C_VEL
LIN {X 0,Y 587.32,Z 282.323,A -85,B 0,C 180,E1 -1285.517,E2 -1285.517} C_VEL
LIN {X 0,Y 587.307,Z 282.322,A -85,B 0,C 180,E1 -1287.82,E2 -1287.82} C_VEL
LIN {X 0,Y 587.321,Z 282.319,A -85,B 0,C 180,E1 -1290.507,E2 -1290.507} C_VEL
LIN {X 0,Y 587.337,Z 282.323,A -85,B 0,C 180,E1 -1293.111,E2 -1293.111} C_VEL
LIN {X 0,Y 587.301,Z 282.331,A -85,B 0,C 180,E1 -1295.538,E2 -1295.538} C_VEL
LIN {X 0,Y 587.322,Z 282.319,A -85,B 0,C 180,E1 -1298.48,E2 -1298.48} C_VEL
LIN {X 0,Y 587.336,Z 282.319,A -85,B 0,C 180,E1 -1301.157,E2 -1301.157} C_VEL
LIN {X 0,Y 587.314,Z 282.325,A -85,B 0,C 180,E1 -1304.112,E2 -1304.112} C_VEL
LIN {X 0,Y 587.305,Z 282.321,A -85,B 0,C 180,E1 -1306.992,E2 -1306.992} C_VEL
LIN {X 0,Y 587.311,Z 282.326,A -85,B 0,C 180,E1 -1309.745,E2 -1309.745} C_VEL
LIN {X 0,Y 587.321,Z 282.325,A -85,B 0,C 180,E1 -1312.39,E2 -1312.39} C_VEL
LIN {X 0,Y 587.319,Z 282.32,A -85,B 0,C 180,E1 -1314.943,E2 -1314.943} C_VEL
LIN {X 0,Y 587.336,Z 282.317,A -85,B 0,C 180,E1 -1317.42,E2 -1317.42} C_VEL
LIN {X 0,Y 587.332,Z 282.319,A -85,B 0,C 180,E1 -1319.829,E2 -1319.829} C_VEL
LIN {X 0,Y 587.342,Z 282.324,A -85,B 0,C 180,E1 -1322.309,E2 -1322.309} C_VEL
LIN {X 0,Y 587.34,Z 282.317,A -85,B 0,C 180,E1 -1325.422,E2 -1325.422} C_VEL
LIN {X 0,Y 587.312,Z 282.323,A -85,B 0,C 180,E1 -1328.225,E2 -1328.225} C_VEL
LIN {X 0,Y 587.337,Z 282.322,A -85,B 0,C 180,E1 -1331.15,E2 -1331.15} C_VEL
LIN {X 0,Y 587.309,Z 282.32,A -85,B 0,C 180,E1 -1334.024,E2 -1334.024} C_VEL
LIN {X 0,Y 587.346,Z 282.316,A -85,B 0,C 180,E1 -1336.153,E2 -1336.153} C_VEL
LIN {X 0,Y 587.338,Z 282.325,A -85,B 0,C 180,E1 -1338.962,E2 -1338.962} C_VEL
LIN {X 0,Y 587.32,Z 282.323,A -85,B 0,C 180,E1 -1341.744,E2 -1341.744} C_VEL
LIN {X 0,Y 587.351,Z 282.318,A -85,B 0,C 180,E1 -1344.442,E2 -1344.442} C_VEL
LIN {X 0,Y 587.522,Z 288.623,A -85,B 0,C 180,E1 -1345.54,E2 -1345.54} C_VEL
LIN {X 0,Y 587.428,Z 306.712,A -85,B 0,C 180,E1 -1348.628,E2 -1348.628} C_VEL
LIN {X 0,Y 587.337,Z 318.148,A -85,B 0,C 180,E1 -1350.556,E2 -1350.556} C_VEL
LIN {X 0,Y 587.884,Z 323.418,A -85,B 0,C 180,E1 -1350.642,E2 -1350.642} C_VEL
LIN {X 0,Y 587.742,Z 425.196,A -85,B 0,C 180,E1 -1351.905,E2 -1351.905} C_VEL
LIN {X 0,Y 587.62,Z 438.258,A -85,B 0,C 180,E1 -1352.206,E2 -1352.206} C_VEL
LIN {X 0,Y 587.592,Z 451.301,A -85,B 0,C 180,E1 -1352.656,E2 -1352.656} C_VEL
LIN {X 0,Y 587.538,Z 462.356,A -85,B 0,C 180,E1 -1353.171,E2 -1353.171} C_VEL
LIN {X 0,Y 587.457,Z 473.858,A -85,B 0,C 180,E1 -1353.858,E2 -1353.858} C_VEL
LIN {X 0,Y 587.38,Z 484.181,A -85,B 0,C 180,E1 -1354.632,E2 -1354.632} C_VEL
LIN {X 0,Y 587.342,Z 491.843,A -85,B 0,C 180,E1 -1355.32,E2 -1355.32} C_VEL
LIN {X 0,Y 587.304,Z 499.881,A -85,B 0,C 180,E1 -1356.182,E2 -1356.182} C_VEL
LIN {X 0,Y 587.222,Z 507.8,A -85,B 0,C 180,E1 -1357.219,E2 -1357.219} C_VEL
LIN {X 0,Y 587.214,Z 514.134,A -85,B 0,C 180,E1 -1358.257,E2 -1358.257} C_VEL
LIN {X 0,Y 587.189,Z 519.193,A -85,B 0,C 180,E1 -1359.298,E2 -1359.298} C_VEL
LIN {X 0,Y 587.17,Z 523.119,A -85,B 0,C 180,E1 -1360.342,E2 -1360.342} C_VEL
LIN {X 0,Y 587.161,Z 525.141,A -85,B 0,C 180,E1 -1361.04,E2 -1361.04} C_VEL
LIN {X 0,Y 587.153,Z 526.742,A -85,B 0,C 180,E1 -1361.74,E2 -1361.74} C_VEL
LIN {X 0,Y 587.159,Z 527.916,A -85,B 0,C 180,E1 -1362.441,E2 -1362.441} C_VEL
LIN {X 0,Y 587.144,Z 528.639,A -85,B 0,C 180,E1 -1363.145,E2 -1363.145} C_VEL
LIN {X 0,Y 587.156,Z 528.976,A -85,B 0,C 180,E1 -1364.18,E2 -1364.18} C_VEL
LIN {X 0,Y 587.13,Z 528.354,A -85,B 0,C 180,E1 -1365.268,E2 -1365.268} C_VEL
LIN {X 0,Y 587.156,Z 527.401,A -85,B 0,C 180,E1 -1365.979,E2 -1365.979} C_VEL
LIN {X 0,Y 587.141,Z 525.907,A -85,B 0,C 180,E1 -1366.747,E2 -1366.747} C_VEL
LIN {X 0,Y 587.16,Z 523.048,A -85,B 0,C 180,E1 -1367.771,E2 -1367.771} C_VEL
LIN {X 0,Y 587.178,Z 518.314,A -85,B 0,C 180,E1 -1368.993,E2 -1368.993} C_VEL
LIN {X 0,Y 587.201,Z 512.47,A -85,B 0,C 180,E1 -1370.126,E2 -1370.126} C_VEL
LIN {X 0,Y 587.26,Z 505.291,A -85,B 0,C 180,E1 -1371.223,E2 -1371.223} C_VEL
LIN {X 0,Y 587.291,Z 497.851,A -85,B 0,C 180,E1 -1372.144,E2 -1372.144} C_VEL
LIN {X 0,Y 587.381,Z 487.892,A -85,B 0,C 180,E1 -1373.14,E2 -1373.14} C_VEL
LIN {X 0,Y 587.417,Z 477.202,A -85,B 0,C 180,E1 -1374.002,E2 -1374.002} C_VEL
LIN {X 0,Y 587.493,Z 466.745,A -85,B 0,C 180,E1 -1374.677,E2 -1374.677} C_VEL
LIN {X 0,Y 587.584,Z 455.157,A -85,B 0,C 180,E1 -1375.267,E2 -1375.267} C_VEL
LIN {X 0,Y 587.63,Z 442.966,A -85,B 0,C 180,E1 -1375.739,E2 -1375.739} C_VEL
LIN {X 0,Y 587.706,Z 429.988,A -85,B 0,C 180,E1 -1376.093,E2 -1376.093} C_VEL
LIN {X 0,Y 587.743,Z 414.798,A -85,B 0,C 180,E1 -1376.33,E2 -1376.33} C_VEL
LIN {X 0,Y 587.707,Z 320.45,A -85,B 0,C 180,E1 -1377.489,E2 -1377.489} C_VEL
LIN {X 0,Y 587.347,Z 318.195,A -85,B 0,C 180,E1 -1377.525,E2 -1377.525} C_VEL
LIN {X 0,Y 587.424,Z 302.577,A -85,B 0,C 180,E1 -1380.164,E2 -1380.164} C_VEL
LIN {X 0,Y 587.523,Z 286.875,A -85,B 0,C 180,E1 -1382.851,E2 -1382.851} C_VEL
LIN {X 0,Y 587.321,Z 282.324,A -85,B 0,C 180,E1 -1383.654,E2 -1383.654} C_VEL
LIN {X 0,Y 587.341,Z 282.327,A -85,B 0,C 180,E1 -1386.746,E2 -1386.746} C_VEL
LIN {X 0,Y 587.315,Z 282.324,A -85,B 0,C 180,E1 -1389.361,E2 -1389.361} C_VEL
LIN {X 0,Y 587.329,Z 282.318,A -85,B 0,C 180,E1 -1392.107,E2 -1392.107} C_VEL
LIN {X 0,Y 587.282,Z 282.335,A -85,B 0,C 180,E1 -1395.086,E2 -1395.086} C_VEL
LIN {X 0,Y 587.295,Z 282.323,A -85,B 0,C 180,E1 -1397.923,E2 -1397.923} C_VEL
LIN {X 0,Y 587.31,Z 282.322,A -85,B 0,C 180,E1 -1400.638,E2 -1400.638} C_VEL
LIN {X 0,Y 587.339,Z 282.328,A -85,B 0,C 180,E1 -1403.292,E2 -1403.292} C_VEL
LIN {X 0,Y 587.323,Z 282.322,A -85,B 0,C 180,E1 -1405.778,E2 -1405.778} C_VEL
LIN {X 0,Y 587.322,Z 282.32,A -85,B 0,C 180,E1 -1408.23,E2 -1408.23} C_VEL
LIN {X 0,Y 587.332,Z 282.318,A -85,B 0,C 180,E1 -1410.868,E2 -1410.868} C_VEL
LIN {X 0,Y 587.292,Z 282.33,A -85,B 0,C 180,E1 -1413.83,E2 -1413.83} C_VEL
LIN {X 0,Y 587.299,Z 282.328,A -85,B 0,C 180,E1 -1415.992,E2 -1415.992} C_VEL
LIN {X 0,Y 587.297,Z 282.325,A -85,B 0,C 180,E1 -1418.225,E2 -1418.225} C_VEL
LIN {X 0,Y 587.314,Z 282.321,A -85,B 0,C 180,E1 -1421.15,E2 -1421.15} C_VEL
LIN {X 0,Y 587.282,Z 282.334,A -85,B 0,C 180,E1 -1424.024,E2 -1424.024} C_VEL
LIN {X 0,Y 587.335,Z 282.325,A -85,B 0,C 180,E1 -1426.154,E2 -1426.154} C_VEL
LIN {X 0,Y 587.279,Z 282.324,A -85,B 0,C 180,E1 -1428.961,E2 -1428.961} C_VEL
LIN {X 0,Y 587.312,Z 282.323,A -85,B 0,C 180,E1 -1431.744,E2 -1431.744} C_VEL
LIN {X 0,Y 587.318,Z 282.326,A -85,B 0,C 180,E1 -1434.507,E2 -1434.507} C_VEL
LIN {X 0,Y 587.314,Z 282.319,A -85,B 0,C 180,E1 -1437.257,E2 -1437.257} C_VEL
LIN {X 0,Y 587.343,Z 282.32,A -85,B 0,C 180,E1 -1440,E2 -1440} C_VEL
LIN {X 0,Y 587.359,Z 282.321,A -85,B 0,C 180,E1 -1442.743,E2 -1442.743} C_VEL
LIN {X 0,Y 587.307,Z 282.321,A -85,B 0,C 180,E1 -1445.494,E2 -1445.494} C_VEL
LIN {X 0,Y 587.291,Z 282.322,A -85,B 0,C 180,E1 -1447.564,E2 -1447.564} C_VEL
LIN {X 0,Y 587.286,Z 282.327,A -85,B 0,C 180,E1 -1450.341,E2 -1450.341} C_VEL
LIN {X 0,Y 587.288,Z 282.328,A -85,B 0,C 180,E1 -1453.143,E2 -1453.143} C_VEL
LIN {X 0,Y 587.285,Z 282.323,A -85,B 0,C 180,E1 -1455.976,E2 -1455.976} C_VEL
LIN {X 0,Y 587.332,Z 282.328,A -85,B 0,C 180,E1 -1459.04,E2 -1459.04} C_VEL
LIN {X 0,Y 587.299,Z 282.322,A -85,B 0,C 180,E1 -1461.775,E2 -1461.775} C_VEL
LIN {X 0,Y 587.294,Z 282.326,A -85,B 0,C 180,E1 -1464.761,E2 -1464.761} C_VEL
LIN {X 0,Y 587.306,Z 282.325,A -85,B 0,C 180,E1 -1467.686,E2 -1467.686} C_VEL
LIN {X 0,Y 587.305,Z 282.321,A -85,B 0,C 180,E1 -1470.172,E2 -1470.172} C_VEL
LIN {X 0,Y 587.319,Z 282.319,A -85,B 0,C 180,E1 -1472.58,E2 -1472.58} C_VEL
LIN {X 0,Y 587.308,Z 282.324,A -85,B 0,C 180,E1 -1475.057,E2 -1475.057} C_VEL
LIN {X 0,Y 587.328,Z 282.324,A -85,B 0,C 180,E1 -1477.839,E2 -1477.839} C_VEL
LIN {X 0,Y 587.301,Z 282.324,A -85,B 0,C 180,E1 -1480.256,E2 -1480.256} C_VEL
LIN {X 0,Y 587.288,Z 282.323,A -85,B 0,C 180,E1 -1483.009,E2 -1483.009} C_VEL
LIN {X 0,Y 587.307,Z 282.332,A -85,B 0,C 180,E1 -1485.889,E2 -1485.889} C_VEL
LIN {X 0,Y 587.326,Z 282.319,A -85,B 0,C 180,E1 -1488.926,E2 -1488.926} C_VEL
LIN {X 0,Y 587.313,Z 282.323,A -85,B 0,C 180,E1 -1491.521,E2 -1491.521} C_VEL
LIN {X 0,Y 587.285,Z 282.335,A -85,B 0,C 180,E1 -1494.101,E2 -1494.101} C_VEL
LIN {X 0,Y 587.33,Z 282.322,A -85,B 0,C 180,E1 -1496.604,E2 -1496.604} C_VEL
LIN {X 0,Y 587.331,Z 282.319,A -85,B 0,C 180,E1 -1499.034,E2 -1499.034} C_VEL
LIN {X 0,Y 587.31,Z 282.321,A -85,B 0,C 180,E1 -1501.403,E2 -1501.403} C_VEL
LIN {X 0,Y 587.328,Z 282.321,A -85,B 0,C 180,E1 -1503.826,E2 -1503.826} C_VEL
LIN {X 0,Y 587.304,Z 282.328,A -85,B 0,C 180,E1 -1505.993,E2 -1505.993} C_VEL
LIN {X 0,Y 587.338,Z 282.455,A -85,B 0,C 180,E1 -1507.261,E2 -1507.261} C_VEL
LIN {X 0,Y 587.801,Z 286.508,A -85,B 0,C 180,E1 -1507.876,E2 -1507.876} C_VEL
LIN {X 0,Y 587.664,Z 306.07,A -85,B 0,C 180,E1 -1510.716,E2 -1510.716} C_VEL
LIN {X 0,Y 587.534,Z 325.547,A -85,B 0,C 180,E1 -1513.496,E2 -1513.496} C_VEL
LIN {X 0,Y 587.404,Z 346.325,A -85,B 0,C 180,E1 -1516.421,E2 -1516.421} C_VEL
LIN {X 0,Y 587.426,Z 347.202,A -85,B 0,C 180,E1 -1516.509,E2 -1516.509} C_VEL
LIN {X 0,Y 587.879,Z 352.568,A -85,B 0,C 180,E1 -1516.586,E2 -1516.586} C_VEL
LIN {X 0,Y 587.724,Z 454.984,A -85,B 0,C 180,E1 -1517.856,E2 -1517.856} C_VEL
LIN {X 0,Y 587.679,Z 468.244,A -85,B 0,C 180,E1 -1518.161,E2 -1518.161} C_VEL
LIN {X 0,Y 587.592,Z 480.62,A -85,B 0,C 180,E1 -1518.584,E2 -1518.584} C_VEL
LIN {X 0,Y 587.552,Z 492.643,A -85,B 0,C 180,E1 -1519.142,E2 -1519.142} C_VEL
LIN {X 0,Y 587.457,Z 504.212,A -85,B 0,C 180,E1 -1519.837,E2 -1519.837} C_VEL
LIN {X 0,Y 587.362,Z 514.547,A -85,B 0,C 180,E1 -1520.618,E2 -1520.618} C_VEL
LIN {X 0,Y 587.298,Z 523.049,A -85,B 0,C 180,E1 -1521.398,E2 -1521.398} C_VEL
LIN {X 0,Y 587.273,Z 530.966,A -85,B 0,C 180,E1 -1522.263,E2 -1522.263} C_VEL
LIN {X 0,Y 587.229,Z 537.474,A -85,B 0,C 180,E1 -1523.127,E2 -1523.127} C_VEL
LIN {X 0,Y 587.236,Z 543.87,A -85,B 0,C 180,E1 -1524.162,E2 -1524.162} C_VEL
LIN {X 0,Y 587.147,Z 548.953,A -85,B 0,C 180,E1 -1525.194,E2 -1525.194} C_VEL
LIN {X 0,Y 587.212,Z 552.898,A -85,B 0,C 180,E1 -1526.226,E2 -1526.226} C_VEL
LIN {X 0,Y 587.132,Z 555.81,A -85,B 0,C 180,E1 -1527.256,E2 -1527.256} C_VEL
LIN {X 0,Y 587.138,Z 557.201,A -85,B 0,C 180,E1 -1527.943,E2 -1527.943} C_VEL
LIN {X 0,Y 587.14,Z 558.785,A -85,B 0,C 180,E1 -1529.315,E2 -1529.315} C_VEL
LIN {X 0,Y 587.137,Z 559,A -85,B 0,C 180,E1 -1530.001,E2 -1530.001} C_VEL
LIN {X 0,Y 587.147,Z 558.185,A -85,B 0,C 180,E1 -1531.372,E2 -1531.372} C_VEL
LIN {X 0,Y 587.138,Z 557.2,A -85,B 0,C 180,E1 -1532.059,E2 -1532.059} C_VEL
LIN {X 0,Y 587.132,Z 555.808,A -85,B 0,C 180,E1 -1532.745,E2 -1532.745} C_VEL
LIN {X 0,Y 587.212,Z 552.894,A -85,B 0,C 180,E1 -1533.775,E2 -1533.775} C_VEL
LIN {X 0,Y 587.147,Z 548.947,A -85,B 0,C 180,E1 -1534.807,E2 -1534.807} C_VEL
LIN {X 0,Y 587.217,Z 542.874,A -85,B 0,C 180,E1 -1536.012,E2 -1536.012} C_VEL
LIN {X 0,Y 587.245,Z 536.233,A -85,B 0,C 180,E1 -1537.047,E2 -1537.047} C_VEL
LIN {X 0,Y 587.298,Z 527.985,A -85,B 0,C 180,E1 -1538.084,E2 -1538.084} C_VEL
LIN {X 0,Y 587.348,Z 519.532,A -85,B 0,C 180,E1 -1538.949,E2 -1538.949} C_VEL
LIN {X 0,Y 587.406,Z 509.088,A -85,B 0,C 180,E1 -1539.817,E2 -1539.817} C_VEL
LIN {X 0,Y 587.501,Z 498.748,A -85,B 0,C 180,E1 -1540.512,E2 -1540.512} C_VEL
LIN {X 0,Y 587.584,Z 486.8,A -85,B 0,C 180,E1 -1541.149,E2 -1541.149} C_VEL
LIN {X 0,Y 587.638,Z 474.58,A -85,B 0,C 180,E1 -1541.64,E2 -1541.64} C_VEL
LIN {X 0,Y 587.684,Z 461.413,A -85,B 0,C 180,E1 -1542.015,E2 -1542.015} C_VEL
LIN {X 0,Y 587.777,Z 449.043,A -85,B 0,C 180,E1 -1542.232,E2 -1542.232} C_VEL
LIN {X 0,Y 587.704,Z 348.889,A -85,B 0,C 180,E1 -1543.463,E2 -1543.463} C_VEL
LIN {X 0,Y 587.381,Z 346.788,A -85,B 0,C 180,E1 -1543.515,E2 -1543.515} C_VEL
LIN {X 0,Y 587.517,Z 328.056,A -85,B 0,C 180,E1 -1546.149,E2 -1546.149} C_VEL
LIN {X 0,Y 587.612,Z 309.166,A -85,B 0,C 180,E1 -1548.841,E2 -1548.841} C_VEL
LIN {X 0,Y 587.776,Z 291.495,A -85,B 0,C 180,E1 -1551.395,E2 -1551.395} C_VEL
LIN {X 0,Y 587.61,Z 283.98,A -85,B 0,C 180,E1 -1552.503,E2 -1552.503} C_VEL
LIN {X 0,Y 587.326,Z 282.326,A -85,B 0,C 180,E1 -1552.79,E2 -1552.79} C_VEL
LIN {X 0,Y 587.335,Z 282.328,A -85,B 0,C 180,E1 -1555.517,E2 -1555.517} C_VEL
LIN {X 0,Y 587.347,Z 282.326,A -85,B 0,C 180,E1 -1557.818,E2 -1557.818} C_VEL
LIN {X 0,Y 587.324,Z 282.319,A -85,B 0,C 180,E1 -1560.507,E2 -1560.507} C_VEL
LIN {X 0,Y 587.336,Z 282.319,A -85,B 0,C 180,E1 -1563.397,E2 -1563.397} C_VEL
LIN {X 0,Y 587.285,Z 282.332,A -85,B 0,C 180,E1 -1565.901,E2 -1565.901} C_VEL
LIN {X 0,Y 587.323,Z 282.323,A -85,B 0,C 180,E1 -1568.48,E2 -1568.48} C_VEL
LIN {X 0,Y 587.334,Z 282.317,A -85,B 0,C 180,E1 -1571.158,E2 -1571.158} C_VEL
LIN {X 0,Y 587.307,Z 282.327,A -85,B 0,C 180,E1 -1574.111,E2 -1574.111} C_VEL
LIN {X 0,Y 587.299,Z 282.324,A -85,B 0,C 180,E1 -1576.992,E2 -1576.992} C_VEL
LIN {X 0,Y 587.311,Z 282.32,A -85,B 0,C 180,E1 -1579.745,E2 -1579.745} C_VEL
LIN {X 0,Y 587.345,Z 282.322,A -85,B 0,C 180,E1 -1582.392,E2 -1582.392} C_VEL
LIN {X 0,Y 587.355,Z 282.314,A -85,B 0,C 180,E1 -1585.779,E2 -1585.779} C_VEL
LIN {X 0,Y 587.335,Z 282.318,A -85,B 0,C 180,E1 -1588.23,E2 -1588.23} C_VEL
LIN {X 0,Y 587.349,Z 282.324,A -85,B 0,C 180,E1 -1590.867,E2 -1590.867} C_VEL
LIN {X 0,Y 587.311,Z 282.321,A -85,B 0,C 180,E1 -1593.72,E2 -1593.72} C_VEL
LIN {X 0,Y 587.296,Z 282.322,A -85,B 0,C 180,E1 -1595.992,E2 -1595.992} C_VEL
LIN {X 0,Y 587.315,Z 282.319,A -85,B 0,C 180,E1 -1598.225,E2 -1598.225} C_VEL
LIN {X 0,Y 587.351,Z 282.322,A -85,B 0,C 180,E1 -1601.151,E2 -1601.151} C_VEL
LIN {X 0,Y 587.315,Z 282.322,A -85,B 0,C 180,E1 -1604.024,E2 -1604.024} C_VEL
LIN {X 0,Y 587.345,Z 282.318,A -85,B 0,C 180,E1 -1606.154,E2 -1606.154} C_VEL
LIN {X 0,Y 587.346,Z 282.316,A -85,B 0,C 180,E1 -1608.962,E2 -1608.962} C_VEL
LIN {X 0,Y 587.329,Z 282.328,A -85,B 0,C 180,E1 -1611.744,E2 -1611.744} C_VEL
LIN {X 0,Y 587.318,Z 282.33,A -85,B 0,C 180,E1 -1613.817,E2 -1613.817} C_VEL
LIN {X 0,Y 587.314,Z 282.33,A -85,B 0,C 180,E1 -1615.883,E2 -1615.883} C_VEL
LIN {X 0,Y 587.376,Z 282.322,A -85,B 0,C 180,E1 -1617.943,E2 -1617.943} C_VEL
LIN {X 0,Y 587.374,Z 282.314,A -85,B 0,C 180,E1 -1620.685,E2 -1620.685} C_VEL
LIN {X 0,Y 587.318,Z 282.319,A -85,B 0,C 180,E1 -1623.43,E2 -1623.43} C_VEL
LIN {X 0,Y 587.316,Z 282.328,A -85,B 0,C 180,E1 -1626.182,E2 -1626.182} C_VEL
LIN {X 0,Y 587.365,Z 282.321,A -85,B 0,C 180,E1 -1628.255,E2 -1628.255} C_VEL
LIN {X 0,Y 587.352,Z 282.317,A -85,B 0,C 180,E1 -1631.133,E2 -1631.133} C_VEL
LIN {X 0,Y 587.367,Z 282.317,A -85,B 0,C 180,E1 -1634.26,E2 -1634.26} C_VEL
LIN {X 0,Y 587.341,Z 282.318,A -85,B 0,C 180,E1 -1637.406,E2 -1637.406} C_VEL
LIN {X 0,Y 587.298,Z 282.324,A -85,B 0,C 180,E1 -1638.301,E2 -1638.301} C_VEL
LIN {X 0,Y 586.663,Z 282.412,A -85,B 0,C 180,E1 -1638.873,E2 -1638.873} C_VEL
LIN {X 0,Y 583.846,Z 282.765,A -85,B 0,C 180,E1 -1639.802,E2 -1639.802} C_VEL
LIN {X 0,Y 581.437,Z 283.064,A -85,B 0,C 180,E1 -1640.549,E2 -1640.549} C_VEL
LIN {X 0,Y 580.381,Z 283.191,A -85,B 0,C 180,E1 -1641.125,E2 -1641.125} C_VEL
LIN {X 0,Y 580.285,Z 283.199,A -85,B 0,C 180,E1 -1641.32,E2 -1641.32} C_VEL
LIN {X 0,Y 580.264,Z 283.2,A -85,B 0,C 180,E1 -1643.558,E2 -1643.558} C_VEL
LIN {X 0,Y 580.272,Z 283.197,A -85,B 0,C 180,E1 -1645.85,E2 -1645.85} C_VEL
LIN {X 0,Y 580.291,Z 283.201,A -85,B 0,C 180,E1 -1648.976,E2 -1648.976} C_VEL
LIN {X 0,Y 580.3,Z 283.194,A -85,B 0,C 180,E1 -1652.03,E2 -1652.03} C_VEL
LIN {X 0,Y 580.293,Z 283.195,A -85,B 0,C 180,E1 -1654.696,E2 -1654.696} C_VEL
LIN {X 0,Y 580.289,Z 283.201,A -85,B 0,C 180,E1 -1657.269,E2 -1657.269} C_VEL
LIN {X 0,Y 580.291,Z 283.196,A -85,B 0,C 180,E1 -1660.27,E2 -1660.27} C_VEL
LIN {X 0,Y 580.26,Z 283.198,A -85,B 0,C 180,E1 -1662.708,E2 -1662.708} C_VEL
LIN {X 0,Y 580.264,Z 283.204,A -85,B 0,C 180,E1 -1665.61,E2 -1665.61} C_VEL
LIN {X 0,Y 580.28,Z 283.202,A -85,B 0,C 180,E1 -1668.231,E2 -1668.231} C_VEL
LIN {X 0,Y 580.268,Z 283.197,A -85,B 0,C 180,E1 -1670.964,E2 -1670.964} C_VEL
LIN {X 0,Y 580.251,Z 283.201,A -85,B 0,C 180,E1 -1673.595,E2 -1673.595} C_VEL
LIN {X 0,Y 580.313,Z 283.201,A -85,B 0,C 180,E1 -1676.145,E2 -1676.145} C_VEL
LIN {X 0,Y 580.274,Z 283.203,A -85,B 0,C 180,E1 -1678.614,E2 -1678.614} C_VEL
LIN {X 0,Y 580.287,Z 283.197,A -85,B 0,C 180,E1 -1681.023,E2 -1681.023} C_VEL
LIN {X 0,Y 580.267,Z 283.198,A -85,B 0,C 180,E1 -1683.671,E2 -1683.671} C_VEL
LIN {X 0,Y 580.261,Z 283.205,A -85,B 0,C 180,E1 -1686.441,E2 -1686.441} C_VEL
LIN {X 0,Y 580.266,Z 283.199,A -85,B 0,C 180,E1 -1689.436,E2 -1689.436} C_VEL
LIN {X 0,Y 580.251,Z 283.2,A -85,B 0,C 180,E1 -1691.644,E2 -1691.644} C_VEL
LIN {X 0,Y 580.259,Z 283.198,A -85,B 0,C 180,E1 -1693.824,E2 -1693.824} C_VEL
LIN {X 0,Y 580.305,Z 283.193,A -85,B 0,C 180,E1 -1695.982,E2 -1695.982} C_VEL
LIN {X 0,Y 580.307,Z 283.198,A -85,B 0,C 180,E1 -1698.826,E2 -1698.826} C_VEL
LIN {X 0,Y 580.295,Z 283.2,A -85,B 0,C 180,E1 -1701.643,E2 -1701.643} C_VEL
LIN {X 0,Y 580.325,Z 283.204,A -85,B 0,C 180,E1 -1704.353,E2 -1704.353} C_VEL
LIN {X 0,Y 580.528,Z 289.639,A -85,B 0,C 180,E1 -1705.486,E2 -1705.486} C_VEL
LIN {X 0,Y 580.409,Z 307.729,A -85,B 0,C 180,E1 -1708.612,E2 -1708.612} C_VEL
LIN {X 0,Y 580.339,Z 318.142,A -85,B 0,C 180,E1 -1710.39,E2 -1710.39} C_VEL
LIN {X 0,Y 580.972,Z 323.164,A -85,B 0,C 180,E1 -1710.476,E2 -1710.476} C_VEL
LIN {X 0,Y 580.814,Z 425.009,A -85,B 0,C 180,E1 -1711.755,E2 -1711.755} C_VEL
LIN {X 0,Y 580.678,Z 437.392,A -85,B 0,C 180,E1 -1712.037,E2 -1712.037} C_VEL
LIN {X 0,Y 580.64,Z 450.113,A -85,B 0,C 180,E1 -1712.471,E2 -1712.471} C_VEL
LIN {X 0,Y 580.543,Z 462.304,A -85,B 0,C 180,E1 -1713.035,E2 -1713.035} C_VEL
LIN {X 0,Y 580.437,Z 473.818,A -85,B 0,C 180,E1 -1713.731,E2 -1713.731} C_VEL
LIN {X 0,Y 580.345,Z 484.167,A -85,B 0,C 180,E1 -1714.514,E2 -1714.514} C_VEL
LIN {X 0,Y 580.294,Z 493.518,A -85,B 0,C 180,E1 -1715.385,E2 -1715.385} C_VEL
LIN {X 0,Y 580.238,Z 501.317,A -85,B 0,C 180,E1 -1716.258,E2 -1716.258} C_VEL
LIN {X 0,Y 580.143,Z 508.911,A -85,B 0,C 180,E1 -1717.307,E2 -1717.307} C_VEL
LIN {X 0,Y 580.132,Z 515.03,A -85,B 0,C 180,E1 -1718.358,E2 -1718.358} C_VEL
LIN {X 0,Y 580.083,Z 519.901,A -85,B 0,C 180,E1 -1719.413,E2 -1719.413} C_VEL
LIN {X 0,Y 580.092,Z 523.647,A -85,B 0,C 180,E1 -1720.47,E2 -1720.47} C_VEL
LIN {X 0,Y 580.071,Z 525.583,A -85,B 0,C 180,E1 -1721.177,E2 -1721.177} C_VEL
LIN {X 0,Y 580.052,Z 527.077,A -85,B 0,C 180,E1 -1721.886,E2 -1721.886} C_VEL
LIN {X 0,Y 580.049,Z 528.118,A -85,B 0,C 180,E1 -1722.596,E2 -1722.596} C_VEL
LIN {X 0,Y 580.059,Z 528.756,A -85,B 0,C 180,E1 -1723.308,E2 -1723.308} C_VEL
LIN {X 0,Y 580.047,Z 528.964,A -85,B 0,C 180,E1 -1724.234,E2 -1724.234} C_VEL
LIN {X 0,Y 580.029,Z 528.157,A -85,B 0,C 180,E1 -1725.459,E2 -1725.459} C_VEL
LIN {X 0,Y 580.064,Z 527.115,A -85,B 0,C 180,E1 -1726.18,E2 -1726.18} C_VEL
LIN {X 0,Y 580.038,Z 525.603,A -85,B 0,C 180,E1 -1726.905,E2 -1726.905} C_VEL
LIN {X 0,Y 580.079,Z 522.454,A -85,B 0,C 180,E1 -1727.995,E2 -1727.995} C_VEL
LIN {X 0,Y 580.094,Z 518.132,A -85,B 0,C 180,E1 -1729.093,E2 -1729.093} C_VEL
LIN {X 0,Y 580.117,Z 512.487,A -85,B 0,C 180,E1 -1730.198,E2 -1730.198} C_VEL
LIN {X 0,Y 580.185,Z 505.311,A -85,B 0,C 180,E1 -1731.308,E2 -1731.308} C_VEL
LIN {X 0,Y 580.228,Z 497.875,A -85,B 0,C 180,E1 -1732.241,E2 -1732.241} C_VEL
LIN {X 0,Y 580.355,Z 488.339,A -85,B 0,C 180,E1 -1733.211,E2 -1733.211} C_VEL
LIN {X 0,Y 580.394,Z 478.504,A -85,B 0,C 180,E1 -1734.026,E2 -1734.026} C_VEL
LIN {X 0,Y 580.503,Z 467.384,A -85,B 0,C 180,E1 -1734.769,E2 -1734.769} C_VEL
LIN {X 0,Y 580.596,Z 455.226,A -85,B 0,C 180,E1 -1735.401,E2 -1735.401} C_VEL
LIN {X 0,Y 580.656,Z 442.003,A -85,B 0,C 180,E1 -1735.915,E2 -1735.915} C_VEL
LIN {X 0,Y 580.738,Z 429.63,A -85,B 0,C 180,E1 -1736.247,E2 -1736.247} C_VEL
LIN {X 0,Y 580.824,Z 414.374,A -85,B 0,C 180,E1 -1736.484,E2 -1736.484} C_VEL
LIN {X 0,Y 580.895,Z 321.753,A -85,B 0,C 180,E1 -1737.634,E2 -1737.634} C_VEL
LIN {X 0,Y 580.327,Z 318.135,A -85,B 0,C 180,E1 -1737.702,E2 -1737.702} C_VEL
LIN {X 0,Y 580.401,Z 303.731,A -85,B 0,C 180,E1 -1740.166,E2 -1740.166} C_VEL
LIN {X 0,Y 580.53,Z 288.504,A -85,B 0,C 180,E1 -1742.802,E2 -1742.802} C_VEL
LIN {X 0,Y 580.281,Z 283.202,A -85,B 0,C 180,E1 -1743.74,E2 -1743.74} C_VEL
LIN {X 0,Y 580.291,Z 283.205,A -85,B 0,C 180,E1 -1746.933,E2 -1746.933} C_VEL
LIN {X 0,Y 580.27,Z 283.198,A -85,B 0,C 180,E1 -1749.934,E2 -1749.934} C_VEL
LIN {X 0,Y 580.265,Z 283.204,A -85,B 0,C 180,E1 -1752.706,E2 -1752.706} C_VEL
LIN {X 0,Y 580.243,Z 283.204,A -85,B 0,C 180,E1 -1755.611,E2 -1755.611} C_VEL
LIN {X 0,Y 580.243,Z 283.201,A -85,B 0,C 180,E1 -1758.228,E2 -1758.228} C_VEL
LIN {X 0,Y 580.258,Z 283.205,A -85,B 0,C 180,E1 -1760.964,E2 -1760.964} C_VEL
LIN {X 0,Y 580.257,Z 283.206,A -85,B 0,C 180,E1 -1763.596,E2 -1763.596} C_VEL
LIN {X 0,Y 580.268,Z 283.196,A -85,B 0,C 180,E1 -1766.142,E2 -1766.142} C_VEL
LIN {X 0,Y 580.255,Z 283.2,A -85,B 0,C 180,E1 -1768.613,E2 -1768.613} C_VEL
LIN {X 0,Y 580.276,Z 283.199,A -85,B 0,C 180,E1 -1771.023,E2 -1771.023} C_VEL
LIN {X 0,Y 580.233,Z 283.205,A -85,B 0,C 180,E1 -1774.148,E2 -1774.148} C_VEL
LIN {X 0,Y 580.249,Z 283.201,A -85,B 0,C 180,E1 -1776.441,E2 -1776.441} C_VEL
LIN {X 0,Y 580.254,Z 283.203,A -85,B 0,C 180,E1 -1779.437,E2 -1779.437} C_VEL
LIN {X 0,Y 580.228,Z 283.209,A -85,B 0,C 180,E1 -1781.644,E2 -1781.644} C_VEL
LIN {X 0,Y 580.254,Z 283.201,A -85,B 0,C 180,E1 -1784.546,E2 -1784.546} C_VEL
LIN {X 0,Y 580.222,Z 283.204,A -85,B 0,C 180,E1 -1786.695,E2 -1786.695} C_VEL
LIN {X 0,Y 580.257,Z 283.2,A -85,B 0,C 180,E1 -1788.826,E2 -1788.826} C_VEL
LIN {X 0,Y 580.278,Z 283.197,A -85,B 0,C 180,E1 -1791.643,E2 -1791.643} C_VEL
LIN {X 0,Y 580.286,Z 283.203,A -85,B 0,C 180,E1 -1794.44,E2 -1794.44} C_VEL
LIN {X 0,Y 580.301,Z 283.196,A -85,B 0,C 180,E1 -1797.918,E2 -1797.918} C_VEL
LIN {X 0,Y 580.347,Z 283.194,A -85,B 0,C 180,E1 -1800.694,E2 -1800.694} C_VEL
LIN {X 0,Y 580.322,Z 283.197,A -85,B 0,C 180,E1 -1802.777,E2 -1802.777} C_VEL
LIN {X 0,Y 580.275,Z 283.197,A -85,B 0,C 180,E1 -1805.56,E2 -1805.56} C_VEL
LIN {X 0,Y 580.242,Z 283.199,A -85,B 0,C 180,E1 -1807.657,E2 -1807.657} C_VEL
LIN {X 0,Y 580.256,Z 283.204,A -85,B 0,C 180,E1 -1810.468,E2 -1810.468} C_VEL
LIN {X 0,Y 580.268,Z 283.204,A -85,B 0,C 180,E1 -1812.592,E2 -1812.592} C_VEL
LIN {X 0,Y 580.264,Z 283.2,A -85,B 0,C 180,E1 -1815.454,E2 -1815.454} C_VEL
LIN {X 0,Y 580.249,Z 283.2,A -85,B 0,C 180,E1 -1817.626,E2 -1817.626} C_VEL
LIN {X 0,Y 580.265,Z 283.198,A -85,B 0,C 180,E1 -1819.824,E2 -1819.824} C_VEL
LIN {X 0,Y 580.243,Z 283.2,A -85,B 0,C 180,E1 -1822.054,E2 -1822.054} C_VEL
LIN {X 0,Y 580.273,Z 283.205,A -85,B 0,C 180,E1 -1825.082,E2 -1825.082} C_VEL
LIN {X 0,Y 580.267,Z 283.197,A -85,B 0,C 180,E1 -1828.187,E2 -1828.187} C_VEL
LIN {X 0,Y 580.261,Z 283.2,A -85,B 0,C 180,E1 -1830.692,E2 -1830.692} C_VEL
LIN {X 0,Y 580.294,Z 283.203,A -85,B 0,C 180,E1 -1833.317,E2 -1833.317} C_VEL
LIN {X 0,Y 580.235,Z 283.209,A -85,B 0,C 180,E1 -1835.756,E2 -1835.756} C_VEL
LIN {X 0,Y 580.277,Z 283.198,A -85,B 0,C 180,E1 -1838.147,E2 -1838.147} C_VEL
LIN {X 0,Y 580.286,Z 283.196,A -85,B 0,C 180,E1 -1840.845,E2 -1840.845} C_VEL
LIN {X 0,Y 580.263,Z 283.206,A -85,B 0,C 180,E1 -1843.66,E2 -1843.66} C_VEL
LIN {X 0,Y 580.261,Z 283.2,A -85,B 0,C 180,E1 -1846.611,E2 -1846.611} C_VEL
LIN {X 0,Y 580.289,Z 283.196,A -85,B 0,C 180,E1 -1849.157,E2 -1849.157} C_VEL
LIN {X 0,Y 580.282,Z 283.206,A -85,B 0,C 180,E1 -1851.928,E2 -1851.928} C_VEL
LIN {X 0,Y 580.246,Z 283.205,A -85,B 0,C 180,E1 -1854.453,E2 -1854.453} C_VEL
LIN {X 0,Y 580.285,Z 283.196,A -85,B 0,C 180,E1 -1856.976,E2 -1856.976} C_VEL
LIN {X 0,Y 580.286,Z 283.196,A -85,B 0,C 180,E1 -1859.426,E2 -1859.426} C_VEL
LIN {X 0,Y 580.292,Z 283.203,A -85,B 0,C 180,E1 -1862.143,E2 -1862.143} C_VEL
LIN {X 0,Y 580.289,Z 283.202,A -85,B 0,C 180,E1 -1864.92,E2 -1864.92} C_VEL
LIN {X 0,Y 580.311,Z 283.357,A -85,B 0,C 180,E1 -1867.107,E2 -1867.107} C_VEL
LIN {X 0,Y 580.876,Z 287.767,A -85,B 0,C 180,E1 -1867.785,E2 -1867.785} C_VEL
LIN {X 0,Y 580.7,Z 306.388,A -85,B 0,C 180,E1 -1870.521,E2 -1870.521} C_VEL
LIN {X 0,Y 580.551,Z 325.547,A -85,B 0,C 180,E1 -1873.292,E2 -1873.292} C_VEL
LIN {X 0,Y 580.399,Z 346.64,A -85,B 0,C 180,E1 -1876.298,E2 -1876.298} C_VEL
LIN {X 0,Y 580.416,Z 347.202,A -85,B 0,C 180,E1 -1876.343,E2 -1876.343} C_VEL
LIN {X 0,Y 580.978,Z 352.568,A -85,B 0,C 180,E1 -1876.424,E2 -1876.424} C_VEL
LIN {X 0,Y 580.809,Z 454.984,A -85,B 0,C 180,E1 -1877.709,E2 -1877.709} C_VEL
LIN {X 0,Y 580.733,Z 468.244,A -85,B 0,C 180,E1 -1878.018,E2 -1878.018} C_VEL
LIN {X 0,Y 580.628,Z 481.15,A -85,B 0,C 180,E1 -1878.466,E2 -1878.466} C_VEL
LIN {X 0,Y 580.561,Z 492.642,A -85,B 0,C 180,E1 -1879.009,E2 -1879.009} C_VEL
LIN {X 0,Y 580.437,Z 504.213,A -85,B 0,C 180,E1 -1879.713,E2 -1879.713} C_VEL
LIN {X 0,Y 580.34,Z 514.562,A -85,B 0,C 180,E1 -1880.503,E2 -1880.503} C_VEL
LIN {X 0,Y 580.262,Z 523.063,A -85,B 0,C 180,E1 -1881.293,E2 -1881.293} C_VEL
LIN {X 0,Y 580.221,Z 530.966,A -85,B 0,C 180,E1 -1882.169,E2 -1882.169} C_VEL
LIN {X 0,Y 580.155,Z 538.641,A -85,B 0,C 180,E1 -1883.22,E2 -1883.22} C_VEL
LIN {X 0,Y 580.139,Z 545.684,A -85,B 0,C 180,E1 -1884.439,E2 -1884.439} C_VEL
LIN {X 0,Y 580.108,Z 550.375,A -85,B 0,C 180,E1 -1885.484,E2 -1885.484} C_VEL
LIN {X 0,Y 580.123,Z 553.959,A -85,B 0,C 180,E1 -1886.528,E2 -1886.528} C_VEL
LIN {X 0,Y 580.043,Z 555.81,A -85,B 0,C 180,E1 -1887.223,E2 -1887.223} C_VEL
LIN {X 0,Y 580.038,Z 557.2,A -85,B 0,C 180,E1 -1887.918,E2 -1887.918} C_VEL
LIN {X 0,Y 580.04,Z 558.785,A -85,B 0,C 180,E1 -1889.306,E2 -1889.306} C_VEL
LIN {X 0,Y 580.037,Z 559,A -85,B 0,C 180,E1 -1890.001,E2 -1890.001} C_VEL
LIN {X 0,Y 580.047,Z 558.185,A -85,B 0,C 180,E1 -1891.389,E2 -1891.389} C_VEL
LIN {X 0,Y 580.038,Z 557.199,A -85,B 0,C 180,E1 -1892.084,E2 -1892.084} C_VEL
LIN {X 0,Y 580.043,Z 555.808,A -85,B 0,C 180,E1 -1892.779,E2 -1892.779} C_VEL
LIN {X 0,Y 580.109,Z 552.894,A -85,B 0,C 180,E1 -1893.821,E2 -1893.821} C_VEL
LIN {X 0,Y 580.054,Z 548.947,A -85,B 0,C 180,E1 -1894.866,E2 -1894.866} C_VEL
LIN {X 0,Y 580.14,Z 542.874,A -85,B 0,C 180,E1 -1896.085,E2 -1896.085} C_VEL
LIN {X 0,Y 580.185,Z 536.233,A -85,B 0,C 180,E1 -1897.133,E2 -1897.133} C_VEL
LIN {X 0,Y 580.246,Z 527.985,A -85,B 0,C 180,E1 -1898.183,E2 -1898.183} C_VEL
LIN {X 0,Y 580.333,Z 517.584,A -85,B 0,C 180,E1 -1899.234,E2 -1899.234} C_VEL
LIN {X 0,Y 580.427,Z 507.919,A -85,B 0,C 180,E1 -1900.024,E2 -1900.024} C_VEL
LIN {X 0,Y 580.533,Z 497.317,A -85,B 0,C 180,E1 -1900.728,E2 -1900.728} C_VEL
LIN {X 0,Y 580.646,Z 485.105,A -85,B 0,C 180,E1 -1901.36,E2 -1901.36} C_VEL
LIN {X 0,Y 580.704,Z 473.157,A -85,B 0,C 180,E1 -1901.829,E2 -1901.829} C_VEL
LIN {X 0,Y 580.764,Z 460.497,A -85,B 0,C 180,E1 -1902.182,E2 -1902.182} C_VEL
LIN {X 0,Y 580.829,Z 447.265,A -85,B 0,C 180,E1 -1902.403,E2 -1902.403} C_VEL
LIN {X 0,Y 580.786,Z 349.559,A -85,B 0,C 180,E1 -1903.618,E2 -1903.618} C_VEL
LIN {X 0,Y 580.383,Z 346.788,A -85,B 0,C 180,E1 -1903.681,E2 -1903.681} C_VEL
LIN {X 0,Y 580.552,Z 325.537,A -85,B 0,C 180,E1 -1906.71,E2 -1906.71} C_VEL
LIN {X 0,Y 580.699,Z 306.382,A -85,B 0,C 180,E1 -1909.479,E2 -1909.479} C_VEL
LIN {X 0,Y 580.902,Z 287.758,A -85,B 0,C 180,E1 -1912.215,E2 -1912.215} C_VEL
LIN {X 0,Y 580.279,Z 283.205,A -85,B 0,C 180,E1 -1912.925,E2 -1912.925} C_VEL
LIN {X 0,Y 580.279,Z 283.204,A -85,B 0,C 180,E1 -1915.85,E2 -1915.85} C_VEL
LIN {X 0,Y 580.296,Z 283.198,A -85,B 0,C 180,E1 -1918.186,E2 -1918.186} C_VEL
LIN {X 0,Y 580.275,Z 283.196,A -85,B 0,C 180,E1 -1920.692,E2 -1920.692} C_VEL
LIN {X 0,Y 580.305,Z 283.194,A -85,B 0,C 180,E1 -1923.316,E2 -1923.316} C_VEL
LIN {X 0,Y 580.236,Z 283.207,A -85,B 0,C 180,E1 -1925.754,E2 -1925.754} C_VEL
LIN {X 0,Y 580.288,Z 283.206,A -85,B 0,C 180,E1 -1928.147,E2 -1928.147} C_VEL
LIN {X 0,Y 580.296,Z 283.195,A -85,B 0,C 180,E1 -1930.844,E2 -1930.844} C_VEL
LIN {X 0,Y 580.242,Z 283.202,A -85,B 0,C 180,E1 -1933.662,E2 -1933.662} C_VEL
LIN {X 0,Y 580.269,Z 283.205,A -85,B 0,C 180,E1 -1936.611,E2 -1936.611} C_VEL
LIN {X 0,Y 580.298,Z 283.195,A -85,B 0,C 180,E1 -1939.156,E2 -1939.156} C_VEL
LIN {X 0,Y 580.289,Z 283.195,A -85,B 0,C 180,E1 -1941.928,E2 -1941.928} C_VEL
LIN {X 0,Y 580.251,Z 283.205,A -85,B 0,C 180,E1 -1944.452,E2 -1944.452} C_VEL
LIN {X 0,Y 580.289,Z 283.203,A -85,B 0,C 180,E1 -1946.975,E2 -1946.975} C_VEL
LIN {X 0,Y 580.284,Z 283.198,A -85,B 0,C 180,E1 -1949.424,E2 -1949.424} C_VEL
LIN {X 0,Y 580.291,Z 283.194,A -85,B 0,C 180,E1 -1952.143,E2 -1952.143} C_VEL
LIN {X 0,Y 580.286,Z 283.202,A -85,B 0,C 180,E1 -1954.919,E2 -1954.919} C_VEL
LIN {X 0,Y 580.26,Z 283.199,A -85,B 0,C 180,E1 -1957.947,E2 -1957.947} C_VEL
LIN {X 0,Y 580.302,Z 283.196,A -85,B 0,C 180,E1 -1960.913,E2 -1960.913} C_VEL
LIN {X 0,Y 580.273,Z 283.202,A -85,B 0,C 180,E1 -1963.825,E2 -1963.825} C_VEL
LIN {X 0,Y 580.316,Z 283.195,A -85,B 0,C 180,E1 -1965.983,E2 -1965.983} C_VEL
LIN {X 0,Y 580.309,Z 283.192,A -85,B 0,C 180,E1 -1968.827,E2 -1968.827} C_VEL
LIN {X 0,Y 580.301,Z 283.202,A -85,B 0,C 180,E1 -1971.643,E2 -1971.643} C_VEL
LIN {X 0,Y 580.278,Z 283.205,A -85,B 0,C 180,E1 -1973.742,E2 -1973.742} C_VEL
LIN {X 0,Y 580.27,Z 283.206,A -85,B 0,C 180,E1 -1975.832,E2 -1975.832} C_VEL
LIN {X 0,Y 580.346,Z 283.197,A -85,B 0,C 180,E1 -1977.918,E2 -1977.918} C_VEL
LIN {X 0,Y 580.347,Z 283.19,A -85,B 0,C 180,E1 -1980.694,E2 -1980.694} C_VEL
LIN {X 0,Y 580.325,Z 283.192,A -85,B 0,C 180,E1 -1982.776,E2 -1982.776} C_VEL
LIN {X 0,Y 580.311,Z 283.193,A -85,B 0,C 180,E1 -1985.56,E2 -1985.56} C_VEL
LIN {X 0,Y 580.327,Z 283.2,A -85,B 0,C 180,E1 -1988.356,E2 -1988.356} C_VEL
LIN {X 0,Y 580.304,Z 283.194,A -85,B 0,C 180,E1 -1991.191,E2 -1991.191} C_VEL
LIN {X 0,Y 580.324,Z 283.192,A -85,B 0,C 180,E1 -1994.017,E2 -1994.017} C_VEL
LIN {X 0,Y 580.316,Z 283.2,A -85,B 0,C 180,E1 -1996.914,E2 -1996.914} C_VEL
LIN {X 0,Y 580.285,Z 283.195,A -85,B 0,C 180,E1 -1999.823,E2 -1999.823} C_VEL
LIN {X 0,Y 580.285,Z 283.199,A -85,B 0,C 180,E1 -2001.32,E2 -2001.32} C_VEL
LIN {X 0,Y 579.582,Z 283.285,A -85,B 0,C 180,E1 -2001.899,E2 -2001.899} C_VEL
LIN {X 0,Y 576.7,Z 283.65,A -85,B 0,C 180,E1 -2002.839,E2 -2002.839} C_VEL
LIN {X 0,Y 574.305,Z 283.943,A -85,B 0,C 180,E1 -2003.595,E2 -2003.595} C_VEL
LIN {X 0,Y 573.309,Z 284.065,A -85,B 0,C 180,E1 -2004.179,E2 -2004.179} C_VEL
LIN {X 0,Y 573.244,Z 284.073,A -85,B 0,C 180,E1 -2004.377,E2 -2004.377} C_VEL
LIN {X 0,Y 573.21,Z 284.085,A -85,B 0,C 180,E1 -2006.978,E2 -2006.978} C_VEL
LIN {X 0,Y 573.239,Z 284.079,A -85,B 0,C 180,E1 -2009.486,E2 -2009.486} C_VEL
LIN {X 0,Y 573.252,Z 284.072,A -85,B 0,C 180,E1 -2012.645,E2 -2012.645} C_VEL
LIN {X 0,Y 573.211,Z 284.082,A -85,B 0,C 180,E1 -2015.187,E2 -2015.187} C_VEL
LIN {X 0,Y 573.23,Z 284.081,A -85,B 0,C 180,E1 -2017.808,E2 -2017.808} C_VEL
LIN {X 0,Y 573.247,Z 284.072,A -85,B 0,C 180,E1 -2020.525,E2 -2020.525} C_VEL
LIN {X 0,Y 573.237,Z 284.082,A -85,B 0,C 180,E1 -2023.668,E2 -2023.668} C_VEL
LIN {X 0,Y 573.231,Z 284.075,A -85,B 0,C 180,E1 -2026.64,E2 -2026.64} C_VEL
LIN {X 0,Y 573.246,Z 284.074,A -85,B 0,C 180,E1 -2029.475,E2 -2029.475} C_VEL
LIN {X 0,Y 573.224,Z 284.085,A -85,B 0,C 180,E1 -2032.191,E2 -2032.191} C_VEL
LIN {X 0,Y 573.233,Z 284.074,A -85,B 0,C 180,E1 -2035.229,E2 -2035.229} C_VEL
LIN {X 0,Y 573.25,Z 284.074,A -85,B 0,C 180,E1 -2037.772,E2 -2037.772} C_VEL
LIN {X 0,Y 573.26,Z 284.078,A -85,B 0,C 180,E1 -2040.633,E2 -2040.633} C_VEL
LIN {X 0,Y 573.209,Z 284.08,A -85,B 0,C 180,E1 -2043.021,E2 -2043.021} C_VEL
LIN {X 0,Y 573.235,Z 284.074,A -85,B 0,C 180,E1 -2045.364,E2 -2045.364} C_VEL
LIN {X 0,Y 573.222,Z 284.075,A -85,B 0,C 180,E1 -2047.661,E2 -2047.661} C_VEL
LIN {X 0,Y 573.236,Z 284.073,A -85,B 0,C 180,E1 -2049.922,E2 -2049.922} C_VEL
LIN {X 0,Y 573.238,Z 284.083,A -85,B 0,C 180,E1 -2052.997,E2 -2052.997} C_VEL
LIN {X 0,Y 573.251,Z 284.072,A -85,B 0,C 180,E1 -2055.806,E2 -2055.806} C_VEL
LIN {X 0,Y 573.264,Z 284.074,A -85,B 0,C 180,E1 -2058.745,E2 -2058.745} C_VEL
LIN {X 0,Y 573.242,Z 284.08,A -85,B 0,C 180,E1 -2061.539,E2 -2061.539} C_VEL
LIN {X 0,Y 573.3,Z 284.103,A -85,B 0,C 180,E1 -2064.261,E2 -2064.261} C_VEL
LIN {X 0,Y 573.491,Z 288.669,A -85,B 0,C 180,E1 -2065.078,E2 -2065.078} C_VEL
LIN {X 0,Y 573.415,Z 302.691,A -85,B 0,C 180,E1 -2067.541,E2 -2067.541} C_VEL
LIN {X 0,Y 573.312,Z 318.141,A -85,B 0,C 180,E1 -2070.219,E2 -2070.219} C_VEL
LIN {X 0,Y 574.089,Z 324.6,A -85,B 0,C 180,E1 -2070.328,E2 -2070.328} C_VEL
LIN {X 0,Y 573.88,Z 424.833,A -85,B 0,C 180,E1 -2071.6,E2 -2071.6} C_VEL
LIN {X 0,Y 573.738,Z 437.273,A -85,B 0,C 180,E1 -2071.886,E2 -2071.886} C_VEL
LIN {X 0,Y 573.667,Z 450.041,A -85,B 0,C 180,E1 -2072.325,E2 -2072.325} C_VEL
LIN {X 0,Y 573.575,Z 462.242,A -85,B 0,C 180,E1 -2072.897,E2 -2072.897} C_VEL
LIN {X 0,Y 573.42,Z 473.779,A -85,B 0,C 180,E1 -2073.601,E2 -2073.601} C_VEL
LIN {X 0,Y 573.316,Z 484.152,A -85,B 0,C 180,E1 -2074.393,E2 -2074.393} C_VEL
LIN {X 0,Y 573.243,Z 493.507,A -85,B 0,C 180,E1 -2075.275,E2 -2075.275} C_VEL
LIN {X 0,Y 573.182,Z 501.295,A -85,B 0,C 180,E1 -2076.158,E2 -2076.158} C_VEL
LIN {X 0,Y 573.066,Z 508.894,A -85,B 0,C 180,E1 -2077.221,E2 -2077.221} C_VEL
LIN {X 0,Y 573.056,Z 515.924,A -85,B 0,C 180,E1 -2078.462,E2 -2078.462} C_VEL
LIN {X 0,Y 572.993,Z 520.606,A -85,B 0,C 180,E1 -2079.53,E2 -2079.53} C_VEL
LIN {X 0,Y 573.008,Z 524.174,A -85,B 0,C 180,E1 -2080.601,E2 -2080.601} C_VEL
LIN {X 0,Y 572.973,Z 525.993,A -85,B 0,C 180,E1 -2081.317,E2 -2081.317} C_VEL
LIN {X 0,Y 572.945,Z 527.358,A -85,B 0,C 180,E1 -2082.035,E2 -2082.035} C_VEL
LIN {X 0,Y 572.944,Z 528.315,A -85,B 0,C 180,E1 -2082.755,E2 -2082.755} C_VEL
LIN {X 0,Y 572.967,Z 528.87,A -85,B 0,C 180,E1 -2083.476,E2 -2083.476} C_VEL
LIN {X 0,Y 572.959,Z 528.95,A -85,B 0,C 180,E1 -2084.298,E2 -2084.298} C_VEL
LIN {X 0,Y 572.931,Z 527.952,A -85,B 0,C 180,E1 -2085.656,E2 -2085.656} C_VEL
LIN {X 0,Y 572.939,Z 525.693,A -85,B 0,C 180,E1 -2086.905,E2 -2086.905} C_VEL
LIN {X 0,Y 572.996,Z 521.818,A -85,B 0,C 180,E1 -2088.225,E2 -2088.225} C_VEL
LIN {X 0,Y 573.039,Z 517.3,A -85,B 0,C 180,E1 -2089.337,E2 -2089.337} C_VEL
LIN {X 0,Y 573.065,Z 511.438,A -85,B 0,C 180,E1 -2090.457,E2 -2090.457} C_VEL
LIN {X 0,Y 573.122,Z 503.964,A -85,B 0,C 180,E1 -2091.584,E2 -2091.584} C_VEL
LIN {X 0,Y 573.191,Z 496.203,A -85,B 0,C 180,E1 -2092.529,E2 -2092.529} C_VEL
LIN {X 0,Y 573.32,Z 487.084,A -85,B 0,C 180,E1 -2093.439,E2 -2093.439} C_VEL
LIN {X 0,Y 573.37,Z 477.273,A -85,B 0,C 180,E1 -2094.243,E2 -2094.243} C_VEL
LIN {X 0,Y 573.496,Z 466.958,A -85,B 0,C 180,E1 -2094.927,E2 -2094.927} C_VEL
LIN {X 0,Y 573.621,Z 455.301,A -85,B 0,C 180,E1 -2095.538,E2 -2095.538} C_VEL
LIN {X 0,Y 573.713,Z 443.167,A -85,B 0,C 180,E1 -2096.02,E2 -2096.02} C_VEL
LIN {X 0,Y 573.806,Z 429.864,A -85,B 0,C 180,E1 -2096.392,E2 -2096.392} C_VEL
LIN {X 0,Y 573.902,Z 415.237,A -85,B 0,C 180,E1 -2096.625,E2 -2096.625} C_VEL
LIN {X 0,Y 574.042,Z 322.708,A -85,B 0,C 180,E1 -2097.787,E2 -2097.787} C_VEL
LIN {X 0,Y 573.296,Z 318.113,A -85,B 0,C 180,E1 -2097.876,E2 -2097.876} C_VEL
LIN {X 0,Y 573.414,Z 302.727,A -85,B 0,C 180,E1 -2100.543,E2 -2100.543} C_VEL
LIN {X 0,Y 573.544,Z 287.298,A -85,B 0,C 180,E1 -2103.253,E2 -2103.253} C_VEL
LIN {X 0,Y 573.231,Z 284.08,A -85,B 0,C 180,E1 -2103.86,E2 -2103.86} C_VEL
LIN {X 0,Y 573.242,Z 284.079,A -85,B 0,C 180,E1 -2107.165,E2 -2107.165} C_VEL
LIN {X 0,Y 573.227,Z 284.077,A -85,B 0,C 180,E1 -2109.608,E2 -2109.608} C_VEL
LIN {X 0,Y 573.23,Z 284.079,A -85,B 0,C 180,E1 -2112.64,E2 -2112.64} C_VEL
LIN {X 0,Y 573.209,Z 284.079,A -85,B 0,C 180,E1 -2115.664,E2 -2115.664} C_VEL
LIN {X 0,Y 573.208,Z 284.079,A -85,B 0,C 180,E1 -2118.541,E2 -2118.541} C_VEL
LIN {X 0,Y 573.225,Z 284.086,A -85,B 0,C 180,E1 -2121.297,E2 -2121.297} C_VEL
LIN {X 0,Y 573.202,Z 284.079,A -85,B 0,C 180,E1 -2124.018,E2 -2124.018} C_VEL
LIN {X 0,Y 573.218,Z 284.073,A -85,B 0,C 180,E1 -2126.515,E2 -2126.515} C_VEL
LIN {X 0,Y 573.208,Z 284.082,A -85,B 0,C 180,E1 -2129.119,E2 -2129.119} C_VEL
LIN {X 0,Y 573.21,Z 284.081,A -85,B 0,C 180,E1 -2131.977,E2 -2131.977} C_VEL
LIN {X 0,Y 573.195,Z 284.078,A -85,B 0,C 180,E1 -2134.587,E2 -2134.587} C_VEL
LIN {X 0,Y 573.226,Z 284.075,A -85,B 0,C 180,E1 -2136.9,E2 -2136.9} C_VEL
LIN {X 0,Y 573.236,Z 284.075,A -85,B 0,C 180,E1 -2139.173,E2 -2139.173} C_VEL
LIN {X 0,Y 573.186,Z 284.083,A -85,B 0,C 180,E1 -2141.41,E2 -2141.41} C_VEL
LIN {X 0,Y 573.194,Z 284.083,A -85,B 0,C 180,E1 -2144.351,E2 -2144.351} C_VEL
LIN {X 0,Y 573.187,Z 284.081,A -85,B 0,C 180,E1 -2146.529,E2 -2146.529} C_VEL
LIN {X 0,Y 573.228,Z 284.075,A -85,B 0,C 180,E1 -2149.403,E2 -2149.403} C_VEL
LIN {X 0,Y 573.206,Z 284.087,A -85,B 0,C 180,E1 -2152.249,E2 -2152.249} C_VEL
LIN {X 0,Y 573.255,Z 284.071,A -85,B 0,C 180,E1 -2155.077,E2 -2155.077} C_VEL
LIN {X 0,Y 573.274,Z 284.071,A -85,B 0,C 180,E1 -2157.892,E2 -2157.892} C_VEL
LIN {X 0,Y 573.317,Z 284.069,A -85,B 0,C 180,E1 -2160.703,E2 -2160.703} C_VEL
LIN {X 0,Y 573.285,Z 284.073,A -85,B 0,C 180,E1 -2162.811,E2 -2162.811} C_VEL
LIN {X 0,Y 573.245,Z 284.072,A -85,B 0,C 180,E1 -2165.629,E2 -2165.629} C_VEL
LIN {X 0,Y 573.2,Z 284.076,A -85,B 0,C 180,E1 -2167.751,E2 -2167.751} C_VEL
LIN {X 0,Y 573.231,Z 284.082,A -85,B 0,C 180,E1 -2170.597,E2 -2170.597} C_VEL
LIN {X 0,Y 573.194,Z 284.079,A -85,B 0,C 180,E1 -2173.472,E2 -2173.472} C_VEL
LIN {X 0,Y 573.214,Z 284.078,A -85,B 0,C 180,E1 -2176.38,E2 -2176.38} C_VEL
LIN {X 0,Y 573.256,Z 284.076,A -85,B 0,C 180,E1 -2179.331,E2 -2179.331} C_VEL
LIN {X 0,Y 573.21,Z 284.077,A -85,B 0,C 180,E1 -2182.339,E2 -2182.339} C_VEL
LIN {X 0,Y 573.222,Z 284.083,A -85,B 0,C 180,E1 -2185.412,E2 -2185.412} C_VEL
LIN {X 0,Y 573.212,Z 284.077,A -85,B 0,C 180,E1 -2188.566,E2 -2188.566} C_VEL
LIN {X 0,Y 573.209,Z 284.081,A -85,B 0,C 180,E1 -2190.995,E2 -2190.995} C_VEL
LIN {X 0,Y 573.256,Z 284.081,A -85,B 0,C 180,E1 -2193.525,E2 -2193.525} C_VEL
LIN {X 0,Y 573.185,Z 284.083,A -85,B 0,C 180,E1 -2196.054,E2 -2196.054} C_VEL
LIN {X 0,Y 573.229,Z 284.074,A -85,B 0,C 180,E1 -2198.703,E2 -2198.703} C_VEL
LIN {X 0,Y 573.219,Z 284.085,A -85,B 0,C 180,E1 -2201.593,E2 -2201.593} C_VEL
LIN {X 0,Y 573.217,Z 284.078,A -85,B 0,C 180,E1 -2204.336,E2 -2204.336} C_VEL
LIN {X 0,Y 573.227,Z 284.078,A -85,B 0,C 180,E1 -2207.36,E2 -2207.36} C_VEL
LIN {X 0,Y 573.232,Z 284.079,A -85,B 0,C 180,E1 -2210.393,E2 -2210.393} C_VEL
LIN {X 0,Y 573.227,Z 284.075,A -85,B 0,C 180,E1 -2213.077,E2 -2213.077} C_VEL
LIN {X 0,Y 573.26,Z 284.074,A -85,B 0,C 180,E1 -2215.672,E2 -2215.672} C_VEL
LIN {X 0,Y 573.242,Z 284.083,A -85,B 0,C 180,E1 -2218.186,E2 -2218.186} C_VEL
LIN {X 0,Y 573.24,Z 284.079,A -85,B 0,C 180,E1 -2220.634,E2 -2220.634} C_VEL
LIN {X 0,Y 573.219,Z 284.079,A -85,B 0,C 180,E1 -2223.023,E2 -2223.023} C_VEL
LIN {X 0,Y 573.235,Z 284.079,A -85,B 0,C 180,E1 -2225.365,E2 -2225.365} C_VEL
LIN {X 0,Y 573.242,Z 284.192,A -85,B 0,C 180,E1 -2226.968,E2 -2226.968} C_VEL
LIN {X 0,Y 573.941,Z 288.898,A -85,B 0,C 180,E1 -2227.692,E2 -2227.692} C_VEL
LIN {X 0,Y 573.765,Z 306.659,A -85,B 0,C 180,E1 -2230.316,E2 -2230.316} C_VEL
LIN {X 0,Y 573.566,Z 325.031,A -85,B 0,C 180,E1 -2233.007,E2 -2233.007} C_VEL
LIN {X 0,Y 573.409,Z 346.325,A -85,B 0,C 180,E1 -2236.083,E2 -2236.083} C_VEL
LIN {X 0,Y 573.422,Z 347.202,A -85,B 0,C 180,E1 -2236.173,E2 -2236.173} C_VEL
